//     Drive/Outputs/Out/nCtrl2 @bit 3 <-> STM Control/Control/Digital output 1
//     Drive/Outputs/Out/nDataOut2[0] <-> STM Velocity/Velocity
//   (this object) <-> Device 2 (EtherCAT)/Rack#2B-01 Coupler (EK1100)/Rack#2B-20 DR_ZF (EL7047)
//     Drive/Inputs/In/nDcOutputTime <-> InfoData/DcOutputShift
//     Drive/Inputs/In/nState1 @bit 3 <-> STM Status/Status/Error
//     Drive/Inputs/In/nState1 @bit 7 <-> STM Status/Status/Motor stall
//     Drive/Inputs/In/nState1 @bit 5 <-> STM Status/Status/Moving negative
//     Drive/Inputs/In/nState1 @bit 4 <-> STM Status/Status/Moving positive
//     Drive/Inputs/In/nState1 @bit 1 <-> STM Status/Status/Ready
//     Drive/Inputs/In/nState1 <-> STM Status/Status/Ready to enable
//     Drive/Inputs/In/nState1 @bit 6 <-> STM Status/Status/Torque reduced
//     Drive/Inputs/In/nState1 @bit 2 <-> STM Status/Status/Warning
//     Drive/Inputs/In/nState2 @bit 3 <-> STM Status/Status/Digital input 1
//     Drive/Inputs/In/nState2 @bit 4 <-> STM Status/Status/Digital input 2
//     Drive/Inputs/In/nState2 @bit 5 <-> STM Status/Status/Sync error
//     Drive/Inputs/In/nState2 @bit 7 <-> STM Status/Status/TxPDO Toggle
//     Drive/Inputs/In/nState4 @bit 1 <-> WcState/InputToggle
//     Drive/Inputs/In/nState4 <-> WcState/WcState
//     Drive/Outputs/Out/nCtrl1 <-> STM Control/Control/Enable
//     Drive/Outputs/Out/nCtrl1 @bit 2 <-> STM Control/Control/Reduce torque
//     Drive/Outputs/Out/nCtrl1 @bit 1 <-> STM Control/Control/Reset
//     Drive/Outputs/Out/nCtrl2 @bit 3 <-> STM Control/Control/Digital output 1
//     Drive/Outputs/Out/nDataOut2[0] <-> STM Velocity/Velocity
//   (this object) <-> Device 2 (EtherCAT)/B950-233-WALL-S-R01-DRL-02/EL5042_03_02-Diff-X-Y
//     Enc/Inputs/In/nComState @bit 1 <-> WcState/InputToggle
//     Enc/Inputs/In/nComState <-> WcState/WcState
//     Enc/Inputs/In/nDataIn1 <-> FB Inputs Channel 2/Position
//     Enc/Inputs/In/nDataIn1 <-> FB Inputs Channel 1/Position
//     Enc/Inputs/In/nState1 @bit 12 <-> FB Inputs Channel 2/Status/Diag
//     Enc/Inputs/In/nState1 @bit 12 <-> FB Inputs Channel 1/Status/Diag
//     Enc/Inputs/In/nState1 @bit 1 <-> FB Inputs Channel 2/Status/Error
//     Enc/Inputs/In/nState1 @bit 1 <-> FB Inputs Channel 1/Status/Error
//     Enc/Inputs/In/nState1 @bit 14 <-> FB Inputs Channel 2/Status/Input cycle counter
//     Enc/Inputs/In/nState1 @bit 14 <-> FB Inputs Channel 1/Status/Input cycle counter
//     Enc/Inputs/In/nState1 @bit 2 <-> FB Inputs Channel 2/Status/Ready
//     Enc/Inputs/In/nState1 @bit 2 <-> FB Inputs Channel 1/Status/Ready
//     Enc/Inputs/In/nState1 @bit 13 <-> FB Inputs Channel 2/Status/TxPDO State
//     Enc/Inputs/In/nState1 @bit 13 <-> FB Inputs Channel 1/Status/TxPDO State
//     Enc/Inputs/In/nState1 <-> FB Inputs Channel 2/Status/Warning
//     Enc/Inputs/In/nState1 <-> FB Inputs Channel 1/Status/Warning
//   (this object) <-> Device 2 (EtherCAT)/B950-233-WALL-S-R01-DRL-02/EL7047_03_03-Diff-Y
//     Drive/Inputs/In/nState1 @bit 3 <-> STM Status/Status/Error
//     Drive/Inputs/In/nState1 @bit 7 <-> STM Status/Status/Motor stall
//     Drive/Inputs/In/nState1 @bit 5 <-> STM Status/Status/Moving negative
//     Drive/Inputs/In/nState1 @bit 4 <-> STM Status/Status/Moving positive
//     Drive/Inputs/In/nState1 @bit 1 <-> STM Status/Status/Ready
//     Drive/Inputs/In/nState1 <-> STM Status/Status/Ready to enable
//     Drive/Inputs/In/nState1 @bit 6 <-> STM Status/Status/Torque reduced
//     Drive/Inputs/In/nState1 @bit 2 <-> STM Status/Status/Warning
//     Drive/Inputs/In/nState2 @bit 3 <-> STM Status/Status/Digital input 1
//     Drive/Inputs/In/nState2 @bit 4 <-> STM Status/Status/Digital input 2
//     Drive/Inputs/In/nState2 @bit 5 <-> STM Status/Status/Sync error
//     Drive/Inputs/In/nState2 @bit 7 <-> STM Status/Status/TxPDO Toggle
//     Drive/Inputs/In/nState4 @bit 1 <-> WcState/InputToggle
//     Drive/Inputs/In/nState4 <-> WcState/WcState
//     Drive/Outputs/Out/nCtrl1 <-> STM Control/Control/Enable
//     Drive/Outputs/Out/nCtrl1 @bit 2 <-> STM Control/Control/Reduce torque
//     Drive/Outputs/Out/nCtrl1 @bit 1 <-> STM Control/Control/Reset
//     Drive/Outputs/Out/nCtrl2 @bit 3 <-> STM Control/Control/Digital output 1
//     Drive/Outputs/Out/nDataOut2[0] <-> STM Velocity/Velocity
//   (this object) <-> Device 2 (EtherCAT)/B950-233-WALL-S-R01-DRL-02/EL5042_03_06-DIff-Z-2ThetaY
//     Enc/Inputs/In/nComState @bit 1 <-> WcState/InputToggle
//     Enc/Inputs/In/nComState <-> WcState/WcState
//     Enc/Inputs/In/nDataIn1 <-> FB Inputs Channel 1/Position
//     Enc/Inputs/In/nDataIn1 <-> FB Inputs Channel 2/Position
//     Enc/Inputs/In/nState1 @bit 12 <-> FB Inputs Channel 1/Status/Diag
//     Enc/Inputs/In/nState1 @bit 12 <-> FB Inputs Channel 2/Status/Diag
//     Enc/Inputs/In/nState1 @bit 1 <-> FB Inputs Channel 1/Status/Error
//     Enc/Inputs/In/nState1 @bit 1 <-> FB Inputs Channel 2/Status/Error
//     Enc/Inputs/In/nState1 @bit 14 <-> FB Inputs Channel 1/Status/Input cycle counter
//     Enc/Inputs/In/nState1 @bit 14 <-> FB Inputs Channel 2/Status/Input cycle counter
//     Enc/Inputs/In/nState1 @bit 2 <-> FB Inputs Channel 1/Status/Ready
//     Enc/Inputs/In/nState1 @bit 2 <-> FB Inputs Channel 2/Status/Ready
//     Enc/Inputs/In/nState1 @bit 13 <-> FB Inputs Channel 1/Status/TxPDO State
//     Enc/Inputs/In/nState1 @bit 13 <-> FB Inputs Channel 2/Status/TxPDO State
//     Enc/Inputs/In/nState1 <-> FB Inputs Channel 1/Status/Warning
//     Enc/Inputs/In/nState1 <-> FB Inputs Channel 2/Status/Warning
//   (this object) <-> Device 2 (EtherCAT)/B950-233-WALL-S-R01-DRL-02/EL7047_03_05-Diff-Z
//     Drive/Inputs/In/nState1 @bit 3 <-> STM Status/Status/Error
//     Drive/Inputs/In/nState1 @bit 7 <-> STM Status/Status/Motor stall
//     Drive/Inputs/In/nState1 @bit 5 <-> STM Status/Status/Moving negative
//     Drive/Inputs/In/nState1 @bit 4 <-> STM Status/Status/Moving positive
//     Drive/Inputs/In/nState1 @bit 1 <-> STM Status/Status/Ready
//     Drive/Inputs/In/nState1 <-> STM Status/Status/Ready to enable
//     Drive/Inputs/In/nState1 @bit 6 <-> STM Status/Status/Torque reduced
//     Drive/Inputs/In/nState1 @bit 2 <-> STM Status/Status/Warning
//     Drive/Inputs/In/nState2 @bit 3 <-> STM Status/Status/Digital input 1
//     Drive/Inputs/In/nState2 @bit 4 <-> STM Status/Status/Digital input 2
//     Drive/Inputs/In/nState2 @bit 5 <-> STM Status/Status/Sync error
//     Drive/Inputs/In/nState2 @bit 7 <-> STM Status/Status/TxPDO Toggle
//     Drive/Inputs/In/nState4 @bit 1 <-> WcState/InputToggle
//     Drive/Inputs/In/nState4 <-> WcState/WcState
//     Drive/Outputs/Out/nCtrl1 <-> STM Control/Control/Enable
//     Drive/Outputs/Out/nCtrl1 @bit 2 <-> STM Control/Control/Reduce torque
//     Drive/Outputs/Out/nCtrl1 @bit 1 <-> STM Control/Control/Reset
//     Drive/Outputs/Out/nCtrl2 @bit 3 <-> STM Control/Control/Digital output 1
//     Drive/Outputs/Out/nDataOut2[0] <-> STM Velocity/Velocity
//   (this object) <-> Device 2 (EtherCAT)/B950-233-WALL-S-R01-DRL-02/EL7047_03_07-Diff 2 Theta Y
//     Drive/Inputs/In/nState1 @bit 3 <-> STM Status/Status/Error
//     Drive/Inputs/In/nState1 @bit 7 <-> STM Status/Status/Motor stall
//     Drive/Inputs/In/nState1 @bit 5 <-> STM Status/Status/Moving negative
//     Drive/Inputs/In/nState1 @bit 4 <-> STM Status/Status/Moving positive
//     Drive/Inputs/In/nState1 @bit 1 <-> STM Status/Status/Ready
//     Drive/Inputs/In/nState1 <-> STM Status/Status/Ready to enable
//     Drive/Inputs/In/nState1 @bit 6 <-> STM Status/Status/Torque reduced
//     Drive/Inputs/In/nState1 @bit 2 <-> STM Status/Status/Warning
//     Drive/Inputs/In/nState2 @bit 3 <-> STM Status/Status/Digital input 1
//     Drive/Inputs/In/nState2 @bit 4 <-> STM Status/Status/Digital input 2
//     Drive/Inputs/In/nState2 @bit 5 <-> STM Status/Status/Sync error
//     Drive/Inputs/In/nState2 @bit 7 <-> STM Status/Status/TxPDO Toggle
//     Drive/Inputs/In/nState4 @bit 1 <-> WcState/InputToggle
//     Drive/Inputs/In/nState4 <-> WcState/WcState
//     Drive/Outputs/Out/nCtrl1 <-> STM Control/Control/Enable
//     Drive/Outputs/Out/nCtrl1 @bit 2 <-> STM Control/Control/Reduce torque
//     Drive/Outputs/Out/nCtrl1 @bit 1 <-> STM Control/Control/Reset
//     Drive/Outputs/Out/nCtrl2 @bit 3 <-> STM Control/Control/Digital output 1
//     Drive/Outputs/Out/nDataOut2[0] <-> STM Velocity/Velocity
//   (this object) <-> Device 2 (EtherCAT)/B950-233-WALL-S-R01-DRL-02/EL5042_03_13 - Diff - Phi - Chi
//     Enc/Inputs/In/nComState @bit 1 <-> WcState/InputToggle
//     Enc/Inputs/In/nComState <-> WcState/WcState
//     Enc/Inputs/In/nDataIn1 <-> FB Inputs Channel 1/Position
//     Enc/Inputs/In/nDataIn1 <-> FB Inputs Channel 2/Position
//     Enc/Inputs/In/nState1 @bit 12 <-> FB Inputs Channel 1/Status/Diag
//     Enc/Inputs/In/nState1 @bit 12 <-> FB Inputs Channel 2/Status/Diag
//     Enc/Inputs/In/nState1 @bit 1 <-> FB Inputs Channel 1/Status/Error
//     Enc/Inputs/In/nState1 @bit 1 <-> FB Inputs Channel 2/Status/Error
//     Enc/Inputs/In/nState1 @bit 14 <-> FB Inputs Channel 1/Status/Input cycle counter
//     Enc/Inputs/In/nState1 @bit 14 <-> FB Inputs Channel 2/Status/Input cycle counter
//     Enc/Inputs/In/nState1 @bit 2 <-> FB Inputs Channel 1/Status/Ready
//     Enc/Inputs/In/nState1 @bit 2 <-> FB Inputs Channel 2/Status/Ready
//     Enc/Inputs/In/nState1 @bit 13 <-> FB Inputs Channel 1/Status/TxPDO State
//     Enc/Inputs/In/nState1 @bit 13 <-> FB Inputs Channel 2/Status/TxPDO State
//     Enc/Inputs/In/nState1 <-> FB Inputs Channel 1/Status/Warning
//     Enc/Inputs/In/nState1 <-> FB Inputs Channel 2/Status/Warning
//   (this object) <-> Device 2 (EtherCAT)/B950-233-WALL-S-R01-DRL-02/EL7047_03_12-Diff - Phi
//     Drive/Inputs/In/nState1 @bit 3 <-> STM Status/Status/Error
//     Drive/Inputs/In/nState1 @bit 7 <-> STM Status/Status/Motor stall
//     Drive/Inputs/In/nState1 @bit 5 <-> STM Status/Status/Moving negative
//     Drive/Inputs/In/nState1 @bit 4 <-> STM Status/Status/Moving positive
//     Drive/Inputs/In/nState1 @bit 1 <-> STM Status/Status/Ready
//     Drive/Inputs/In/nState1 <-> STM Status/Status/Ready to enable
//     Drive/Inputs/In/nState1 @bit 6 <-> STM Status/Status/Torque reduced
//     Drive/Inputs/In/nState1 @bit 2 <-> STM Status/Status/Warning
//     Drive/Inputs/In/nState2 @bit 3 <-> STM Status/Status/Digital input 1
//     Drive/Inputs/In/nState2 @bit 4 <-> STM Status/Status/Digital input 2
//     Drive/Inputs/In/nState2 @bit 5 <-> STM Status/Status/Sync error
//     Drive/Inputs/In/nState2 @bit 7 <-> STM Status/Status/TxPDO Toggle
//     Drive/Inputs/In/nState4 @bit 1 <-> WcState/InputToggle
//     Drive/Inputs/In/nState4 <-> WcState/WcState
//     Drive/Outputs/Out/nCtrl1 <-> STM Control/Control/Enable
//     Drive/Outputs/Out/nCtrl1 @bit 2 <-> STM Control/Control/Reduce torque
//     Drive/Outputs/Out/nCtrl1 @bit 1 <-> STM Control/Control/Reset
//     Drive/Outputs/Out/nCtrl2 @bit 3 <-> STM Control/Control/Digital output 1
//     Drive/Outputs/Out/nDataOut2[0] <-> STM Velocity/Velocity
//   (this object) <-> Device 2 (EtherCAT)/B950-233-WALL-S-R01-DRL-02/EL7047_03_14-Diff - Chi
//     Drive/Inputs/In/nState1 @bit 3 <-> STM Status/Status/Error
//     Drive/Inputs/In/nState1 @bit 7 <-> STM Status/Status/Motor stall
//     Drive/Inputs/In/nState1 @bit 5 <-> STM Status/Status/Moving negative
//     Drive/Inputs/In/nState1 @bit 4 <-> STM Status/Status/Moving positive
//     Drive/Inputs/In/nState1 @bit 1 <-> STM Status/Status/Ready
//     Drive/Inputs/In/nState1 <-> STM Status/Status/Ready to enable
//     Drive/Inputs/In/nState1 @bit 6 <-> STM Status/Status/Torque reduced
//     Drive/Inputs/In/nState1 @bit 2 <-> STM Status/Status/Warning
//     Drive/Inputs/In/nState2 @bit 3 <-> STM Status/Status/Digital input 1
//     Drive/Inputs/In/nState2 @bit 4 <-> STM Status/Status/Digital input 2
//     Drive/Inputs/In/nState2 @bit 5 <-> STM Status/Status/Sync error
//     Drive/Inputs/In/nState2 @bit 7 <-> STM Status/Status/TxPDO Toggle
//     Drive/Inputs/In/nState4 @bit 1 <-> WcState/InputToggle
//     Drive/Inputs/In/nState4 <-> WcState/WcState
//     Drive/Outputs/Out/nCtrl1 <-> STM Control/Control/Enable
//     Drive/Outputs/Out/nCtrl1 @bit 2 <-> STM Control/Control/Reduce torque
//     Drive/Outputs/Out/nCtrl1 @bit 1 <-> STM Control/Control/Reset
//     Drive/Outputs/Out/nCtrl2 @bit 3 <-> STM Control/Control/Digital output 1
//     Drive/Outputs/Out/nDataOut2[0] <-> STM Velocity/Velocity
//   (this object) <-> Device 2 (EtherCAT)/B950-233-WALL-S-R01-DRL-02/EL5042_03_17 - Diff - Theta - 2Theta
//     Enc/Inputs/In/nComState @bit 1 <-> WcState/InputToggle
//     Enc/Inputs/In/nComState <-> WcState/WcState
//     Enc/Inputs/In/nDataIn1 <-> FB Inputs Channel 2/Position
//     Enc/Inputs/In/nState1 @bit 12 <-> FB Inputs Channel 2/Status/Diag
//     Enc/Inputs/In/nState1 @bit 12 <-> FB Inputs Channel 1/Status/Diag
//     Enc/Inputs/In/nState1 @bit 1 <-> FB Inputs Channel 2/Status/Error
//     Enc/Inputs/In/nState1 @bit 1 <-> FB Inputs Channel 1/Status/Error
//     Enc/Inputs/In/nState1 @bit 14 <-> FB Inputs Channel 2/Status/Input cycle counter
//     Enc/Inputs/In/nState1 @bit 14 <-> FB Inputs Channel 1/Status/Input cycle counter
//     Enc/Inputs/In/nState1 @bit 2 <-> FB Inputs Channel 2/Status/Ready
//     Enc/Inputs/In/nState1 @bit 2 <-> FB Inputs Channel 1/Status/Ready
//     Enc/Inputs/In/nState1 @bit 13 <-> FB Inputs Channel 2/Status/TxPDO State
//     Enc/Inputs/In/nState1 @bit 13 <-> FB Inputs Channel 1/Status/TxPDO State
//     Enc/Inputs/In/nState1 <-> FB Inputs Channel 2/Status/Warning
//     Enc/Inputs/In/nState1 <-> FB Inputs Channel 1/Status/Warning
//   (this object) <-> Device 2 (EtherCAT)/B950-233-WALL-S-R01-DRL-02/EL7047_03_18 - Diff - 2Theta
//     Drive/Inputs/In/nState1 @bit 3 <-> STM Status/Status/Error
//     Drive/Inputs/In/nState1 @bit 7 <-> STM Status/Status/Motor stall
//     Drive/Inputs/In/nState1 @bit 5 <-> STM Status/Status/Moving negative
//     Drive/Inputs/In/nState1 @bit 4 <-> STM Status/Status/Moving positive
//     Drive/Inputs/In/nState1 @bit 1 <-> STM Status/Status/Ready
//     Drive/Inputs/In/nState1 <-> STM Status/Status/Ready to enable
//     Drive/Inputs/In/nState1 @bit 6 <-> STM Status/Status/Torque reduced
//     Drive/Inputs/In/nState1 @bit 2 <-> STM Status/Status/Warning
//     Drive/Inputs/In/nState2 @bit 3 <-> STM Status/Status/Digital input 1
//     Drive/Inputs/In/nState2 @bit 4 <-> STM Status/Status/Digital input 2
//     Drive/Inputs/In/nState2 @bit 5 <-> STM Status/Status/Sync error
//     Drive/Inputs/In/nState2 @bit 7 <-> STM Status/Status/TxPDO Toggle
//     Drive/Inputs/In/nState4 @bit 1 <-> WcState/InputToggle
//     Drive/Inputs/In/nState4 <-> WcState/WcState
//     Drive/Outputs/Out/nCtrl1 <-> STM Control/Control/Enable
//     Drive/Outputs/Out/nCtrl1 @bit 2 <-> STM Control/Control/Reduce torque
//     Drive/Outputs/Out/nCtrl1 @bit 1 <-> STM Control/Control/Reset
//     Drive/Outputs/Out/nCtrl2 @bit 3 <-> STM Control/Control/Digital output 1
//     Drive/Outputs/Out/nDataOut2[0] <-> STM Velocity/Velocity
//   (this object) <-> Device 2 (EtherCAT)/B950-233-WALL-S-R01-DRL-02/EL7047_03_16 - Diff - Theta
//     Drive/Inputs/In/nState1 @bit 3 <-> STM Status/Status/Error
//     Drive/Inputs/In/nState1 @bit 7 <-> STM Status/Status/Motor stall
//     Drive/Inputs/In/nState1 @bit 5 <-> STM Status/Status/Moving negative
//     Drive/Inputs/In/nState1 @bit 4 <-> STM Status/Status/Moving positive
//     Drive/Inputs/In/nState1 @bit 1 <-> STM Status/Status/Ready
//     Drive/Inputs/In/nState1 <-> STM Status/Status/Ready to enable
//     Drive/Inputs/In/nState1 @bit 6 <-> STM Status/Status/Torque reduced
//     Drive/Inputs/In/nState1 @bit 2 <-> STM Status/Status/Warning
//     Drive/Inputs/In/nState2 @bit 3 <-> STM Status/Status/Digital input 1
//     Drive/Inputs/In/nState2 @bit 4 <-> STM Status/Status/Digital input 2
//     Drive/Inputs/In/nState2 @bit 5 <-> STM Status/Status/Sync error
//     Drive/Inputs/In/nState2 @bit 7 <-> STM Status/Status/TxPDO Toggle
//     Drive/Inputs/In/nState4 @bit 1 <-> WcState/InputToggle
//     Drive/Inputs/In/nState4 <-> WcState/WcState
//     Drive/Outputs/Out/nCtrl1 <-> STM Control/Control/Enable
//     Drive/Outputs/Out/nCtrl1 @bit 2 <-> STM Control/Control/Reduce torque
//     Drive/Outputs/Out/nCtrl1 @bit 1 <-> STM Control/Control/Reset
//     Drive/Outputs/Out/nCtrl2 @bit 3 <-> STM Control/Control/Digital output 1
//     Drive/Outputs/Out/nDataOut2[0] <-> STM Velocity/Velocity
//   (this object) <-> Device 2 (EtherCAT)/B950-233-WALL-S-R01-DRL-02/EL7047_03_01-Diff-X
//     Drive/Inputs/In/nState1 @bit 3 <-> STM Status/Status/Error
//     Drive/Inputs/In/nState1 @bit 7 <-> STM Status/Status/Motor stall
//     Drive/Inputs/In/nState1 @bit 5 <-> STM Status/Status/Moving negative
//     Drive/Inputs/In/nState1 @bit 4 <-> STM Status/Status/Moving positive
//     Drive/Inputs/In/nState1 @bit 1 <-> STM Status/Status/Ready
//     Drive/Inputs/In/nState1 <-> STM Status/Status/Ready to enable
//     Drive/Inputs/In/nState1 @bit 6 <-> STM Status/Status/Torque reduced
//     Drive/Inputs/In/nState1 @bit 2 <-> STM Status/Status/Warning
//     Drive/Inputs/In/nState2 @bit 3 <-> STM Status/Status/Digital input 1
//     Drive/Inputs/In/nState2 @bit 4 <-> STM Status/Status/Digital input 2
//     Drive/Inputs/In/nState2 @bit 5 <-> STM Status/Status/Sync error
//     Drive/Inputs/In/nState2 @bit 7 <-> STM Status/Status/TxPDO Toggle
//     Drive/Inputs/In/nState4 @bit 1 <-> WcState/InputToggle
//     Drive/Inputs/In/nState4 <-> WcState/WcState
//     Drive/Outputs/Out/nCtrl1 <-> STM Control/Control/Enable
//     Drive/Outputs/Out/nCtrl1 @bit 2 <-> STM Control/Control/Reduce torque
//     Drive/Outputs/Out/nCtrl1 @bit 1 <-> STM Control/Control/Reset
//     Drive/Outputs/Out/nCtrl2 @bit 3 <-> STM Control/Control/Digital output 1
//     Drive/Outputs/Out/nDataOut2[0] <-> STM Velocity/Velocity
//   (this object) <-> Device 2 (EtherCAT)/B950-233-WALL-S-R01-DRL-01/EL5042_02_05 - LAS_VIS
//     Enc/Inputs/In/nComState @bit 1 <-> WcState/InputToggle
//     Enc/Inputs/In/nComState <-> WcState/WcState
//     Enc/Inputs/In/nDataIn1 <-> FB Inputs Channel 1/Position
//     Enc/Inputs/In/nState1 @bit 12 <-> FB Inputs Channel 1/Status/Diag
//     Enc/Inputs/In/nState1 @bit 1 <-> FB Inputs Channel 1/Status/Error
//     Enc/Inputs/In/nState1 @bit 14 <-> FB Inputs Channel 1/Status/Input cycle counter
//     Enc/Inputs/In/nState1 @bit 2 <-> FB Inputs Channel 1/Status/Ready
//     Enc/Inputs/In/nState1 @bit 13 <-> FB Inputs Channel 1/Status/TxPDO State
//     Enc/Inputs/In/nState1 <-> FB Inputs Channel 1/Status/Warning
//   (this object) <-> Device 2 (EtherCAT)/B950-233-WALL-S-R01-DRL-01/EL7031_02_04 - LAS_VIS
//     Drive/Inputs/In/nState1 @bit 3 <-> STM Status/Status/Error
//     Drive/Inputs/In/nState1 @bit 5 <-> STM Status/Status/Moving negative
//     Drive/Inputs/In/nState1 @bit 4 <-> STM Status/Status/Moving positive
//     Drive/Inputs/In/nState1 @bit 1 <-> STM Status/Status/Ready
//     Drive/Inputs/In/nState1 <-> STM Status/Status/Ready to enable
//     Drive/Inputs/In/nState1 @bit 6 <-> STM Status/Status/Torque reduced
//     Drive/Inputs/In/nState1 @bit 2 <-> STM Status/Status/Warning
//     Drive/Inputs/In/nState2 @bit 3 <-> STM Status/Status/Digital input 1
//     Drive/Inputs/In/nState2 @bit 4 <-> STM Status/Status/Digital input 2
//     Drive/Inputs/In/nState2 @bit 5 <-> STM Status/Status/Sync error
//     Drive/Inputs/In/nState2 @bit 7 <-> STM Status/Status/TxPDO Toggle
//     Drive/Inputs/In/nState4 @bit 1 <-> WcState/InputToggle
//     Drive/Inputs/In/nState4 <-> WcState/WcState
//     Drive/Outputs/Out/nCtrl1 <-> STM Control/Control/Enable
//     Drive/Outputs/Out/nCtrl1 @bit 2 <-> STM Control/Control/Reduce torque
//     Drive/Outputs/Out/nCtrl1 @bit 1 <-> STM Control/Control/Reset
//     Drive/Outputs/Out/nDataOut2[0] <-> STM Velocity/Velocity
//   (this object) <-> Device 2 (EtherCAT)/B950-233-WALL-S-R01-DRL-01/EL5042_02_08 - LAS_D_V-H
//     Enc/Inputs/In/nComState @bit 1 <-> WcState/InputToggle
//     Enc/Inputs/In/nComState <-> WcState/WcState
//     Enc/Inputs/In/nDataIn1 <-> FB Inputs Channel 2/Position
//     Enc/Inputs/In/nDataIn1 <-> FB Inputs Channel 1/Position
//     Enc/Inputs/In/nState1 @bit 12 <-> FB Inputs Channel 2/Status/Diag
//     Enc/Inputs/In/nState1 @bit 12 <-> FB Inputs Channel 1/Status/Diag
//     Enc/Inputs/In/nState1 @bit 1 <-> FB Inputs Channel 2/Status/Error
//     Enc/Inputs/In/nState1 @bit 1 <-> FB Inputs Channel 1/Status/Error
//     Enc/Inputs/In/nState1 @bit 14 <-> FB Inputs Channel 2/Status/Input cycle counter
//     Enc/Inputs/In/nState1 @bit 14 <-> FB Inputs Channel 1/Status/Input cycle counter
//     Enc/Inputs/In/nState1 @bit 2 <-> FB Inputs Channel 2/Status/Ready
//     Enc/Inputs/In/nState1 @bit 2 <-> FB Inputs Channel 1/Status/Ready
//     Enc/Inputs/In/nState1 @bit 13 <-> FB Inputs Channel 2/Status/TxPDO State
//     Enc/Inputs/In/nState1 @bit 13 <-> FB Inputs Channel 1/Status/TxPDO State
//     Enc/Inputs/In/nState1 <-> FB Inputs Channel 2/Status/Warning
//     Enc/Inputs/In/nState1 <-> FB Inputs Channel 1/Status/Warning
//   (this object) <-> Device 2 (EtherCAT)/B950-233-WALL-S-R01-DRL-01/EL7031_02_07 - LAS_D_H
//     Drive/Inputs/In/nState1 @bit 3 <-> STM Status/Status/Error
//     Drive/Inputs/In/nState1 @bit 5 <-> STM Status/Status/Moving negative
//     Drive/Inputs/In/nState1 @bit 4 <-> STM Status/Status/Moving positive
//     Drive/Inputs/In/nState1 @bit 1 <-> STM Status/Status/Ready
//     Drive/Inputs/In/nState1 <-> STM Status/Status/Ready to enable
//     Drive/Inputs/In/nState1 @bit 6 <-> STM Status/Status/Torque reduced
//     Drive/Inputs/In/nState1 @bit 2 <-> STM Status/Status/Warning
//     Drive/Inputs/In/nState2 @bit 3 <-> STM Status/Status/Digital input 1
//     Drive/Inputs/In/nState2 @bit 4 <-> STM Status/Status/Digital input 2
//     Drive/Inputs/In/nState2 @bit 5 <-> STM Status/Status/Sync error
//     Drive/Inputs/In/nState2 @bit 7 <-> STM Status/Status/TxPDO Toggle
//     Drive/Inputs/In/nState4 @bit 1 <-> WcState/InputToggle
//     Drive/Inputs/In/nState4 <-> WcState/WcState
//     Drive/Outputs/Out/nCtrl1 <-> STM Control/Control/Enable
//     Drive/Outputs/Out/nCtrl1 @bit 2 <-> STM Control/Control/Reduce torque
//     Drive/Outputs/Out/nCtrl1 @bit 1 <-> STM Control/Control/Reset
//     Drive/Outputs/Out/nDataOut2[0] <-> STM Velocity/Velocity
//   (this object) <-> Device 2 (EtherCAT)/B950-233-WALL-S-R01-DRL-01/EL7031_02_09 - LAS_D_V
//     Drive/Inputs/In/nState1 @bit 3 <-> STM Status/Status/Error
//     Drive/Inputs/In/nState1 @bit 5 <-> STM Status/Status/Moving negative
//     Drive/Inputs/In/nState1 @bit 4 <-> STM Status/Status/Moving positive
//     Drive/Inputs/In/nState1 @bit 1 <-> STM Status/Status/Ready
//     Drive/Inputs/In/nState1 <-> STM Status/Status/Ready to enable
//     Drive/Inputs/In/nState1 @bit 6 <-> STM Status/Status/Torque reduced
//     Drive/Inputs/In/nState1 @bit 2 <-> STM Status/Status/Warning
//     Drive/Inputs/In/nState2 @bit 3 <-> STM Status/Status/Digital input 1
//     Drive/Inputs/In/nState2 @bit 4 <-> STM Status/Status/Digital input 2
//     Drive/Inputs/In/nState2 @bit 5 <-> STM Status/Status/Sync error
//     Drive/Inputs/In/nState2 @bit 7 <-> STM Status/Status/TxPDO Toggle
//     Drive/Inputs/In/nState4 @bit 1 <-> WcState/InputToggle
//     Drive/Inputs/In/nState4 <-> WcState/WcState
//     Drive/Outputs/Out/nCtrl1 <-> STM Control/Control/Enable
//     Drive/Outputs/Out/nCtrl1 @bit 2 <-> STM Control/Control/Reduce torque
//     Drive/Outputs/Out/nCtrl1 @bit 1 <-> STM Control/Control/Reset
//     Drive/Outputs/Out/nDataOut2[0] <-> STM Velocity/Velocity
//   (this object) <-> Device 2 (EtherCAT)/B950-233-WALL-S-R01-DRL-03_SDS/EL5042_04_02
//     Enc/Inputs/In/nComState @bit 1 <-> WcState/InputToggle
//     Enc/Inputs/In/nComState <-> WcState/WcState
//     Enc/Inputs/In/nDataIn1 <-> FB Inputs Channel 1/Position
//     Enc/Inputs/In/nDataIn1 <-> FB Inputs Channel 2/Position
//     Enc/Inputs/In/nState1 @bit 12 <-> FB Inputs Channel 1/Status/Diag
//     Enc/Inputs/In/nState1 @bit 12 <-> FB Inputs Channel 2/Status/Diag
//     Enc/Inputs/In/nState1 @bit 1 <-> FB Inputs Channel 1/Status/Error
//     Enc/Inputs/In/nState1 @bit 1 <-> FB Inputs Channel 2/Status/Error
//     Enc/Inputs/In/nState1 @bit 14 <-> FB Inputs Channel 1/Status/Input cycle counter
//     Enc/Inputs/In/nState1 @bit 14 <-> FB Inputs Channel 2/Status/Input cycle counter
//     Enc/Inputs/In/nState1 @bit 2 <-> FB Inputs Channel 1/Status/Ready
//     Enc/Inputs/In/nState1 @bit 2 <-> FB Inputs Channel 2/Status/Ready
//     Enc/Inputs/In/nState1 @bit 13 <-> FB Inputs Channel 1/Status/TxPDO State
//     Enc/Inputs/In/nState1 @bit 13 <-> FB Inputs Channel 2/Status/TxPDO State
//     Enc/Inputs/In/nState1 <-> FB Inputs Channel 1/Status/Warning
//     Enc/Inputs/In/nState1 <-> FB Inputs Channel 2/Status/Warning
//   (this object) <-> Device 2 (EtherCAT)/B950-233-WALL-S-R01-DRL-03_SDS/EL7047_04_01
//     Drive/Inputs/In/nState1 @bit 3 <-> STM Status/Status/Error
//     Drive/Inputs/In/nState1 @bit 7 <-> STM Status/Status/Motor stall
//     Drive/Inputs/In/nState1 @bit 5 <-> STM Status/Status/Moving negative
//     Drive/Inputs/In/nState1 @bit 4 <-> STM Status/Status/Moving positive
//     Drive/Inputs/In/nState1 @bit 1 <-> STM Status/Status/Ready
//     Drive/Inputs/In/nState1 <-> STM Status/Status/Ready to enable
//     Drive/Inputs/In/nState1 @bit 6 <-> STM Status/Status/Torque reduced
//     Drive/Inputs/In/nState1 @bit 2 <-> STM Status/Status/Warning
//     Drive/Inputs/In/nState2 @bit 3 <-> STM Status/Status/Digital input 1
//     Drive/Inputs/In/nState2 @bit 4 <-> STM Status/Status/Digital input 2
//     Drive/Inputs/In/nState2 @bit 5 <-> STM Status/Status/Sync error
//     Drive/Inputs/In/nState2 @bit 7 <-> STM Status/Status/TxPDO Toggle
//     Drive/Inputs/In/nState4 @bit 1 <-> WcState/InputToggle
//     Drive/Inputs/In/nState4 <-> WcState/WcState
//     Drive/Outputs/Out/nCtrl1 <-> STM Control/Control/Enable
//     Drive/Outputs/Out/nCtrl1 @bit 2 <-> STM Control/Control/Reduce torque
//     Drive/Outputs/Out/nCtrl1 @bit 1 <-> STM Control/Control/Reset
//     Drive/Outputs/Out/nCtrl2 @bit 3 <-> STM Control/Control/Digital output 1
//     Drive/Outputs/Out/nDataOut2[0] <-> STM Velocity/Velocity
//   (this object) <-> Device 2 (EtherCAT)/B950-233-WALL-S-R01-DRL-03_SDS/EL7047_04_03
//     Drive/Inputs/In/nState1 @bit 3 <-> STM Status/Status/Error
//     Drive/Inputs/In/nState1 @bit 7 <-> STM Status/Status/Motor stall
//     Drive/Inputs/In/nState1 @bit 5 <-> STM Status/Status/Moving negative
//     Drive/Inputs/In/nState1 @bit 4 <-> STM Status/Status/Moving positive
//     Drive/Inputs/In/nState1 @bit 1 <-> STM Status/Status/Ready
//     Drive/Inputs/In/nState1 <-> STM Status/Status/Ready to enable
//     Drive/Inputs/In/nState1 @bit 6 <-> STM Status/Status/Torque reduced
//     Drive/Inputs/In/nState1 @bit 2 <-> STM Status/Status/Warning
//     Drive/Inputs/In/nState2 @bit 3 <-> STM Status/Status/Digital input 1
//     Drive/Inputs/In/nState2 @bit 4 <-> STM Status/Status/Digital input 2
//     Drive/Inputs/In/nState2 @bit 5 <-> STM Status/Status/Sync error
//     Drive/Inputs/In/nState2 @bit 7 <-> STM Status/Status/TxPDO Toggle
//     Drive/Inputs/In/nState4 @bit 1 <-> WcState/InputToggle
//     Drive/Inputs/In/nState4 <-> WcState/WcState
//     Drive/Outputs/Out/nCtrl1 <-> STM Control/Control/Enable
//     Drive/Outputs/Out/nCtrl1 @bit 2 <-> STM Control/Control/Reduce torque
//     Drive/Outputs/Out/nCtrl1 @bit 1 <-> STM Control/Control/Reset
//     Drive/Outputs/Out/nCtrl2 @bit 3 <-> STM Control/Control/Digital output 1
//     Drive/Outputs/Out/nDataOut2[0] <-> STM Velocity/Velocity
//   (this object) <-> Device 2 (EtherCAT)/B950-233-WALL-S-R01-DRL-03_SDS/EL5042_04_06
//     Enc/Inputs/In/nComState @bit 1 <-> WcState/InputToggle
//     Enc/Inputs/In/nComState <-> WcState/WcState
//     Enc/Inputs/In/nDataIn1 <-> FB Inputs Channel 1/Position
//     Enc/Inputs/In/nState1 @bit 12 <-> FB Inputs Channel 1/Status/Diag
//     Enc/Inputs/In/nState1 @bit 1 <-> FB Inputs Channel 1/Status/Error
//     Enc/Inputs/In/nState1 @bit 14 <-> FB Inputs Channel 1/Status/Input cycle counter
//     Enc/Inputs/In/nState1 @bit 2 <-> FB Inputs Channel 1/Status/Ready
//     Enc/Inputs/In/nState1 @bit 13 <-> FB Inputs Channel 1/Status/TxPDO State
//     Enc/Inputs/In/nState1 <-> FB Inputs Channel 1/Status/Warning
//   (this object) <-> Device 2 (EtherCAT)/B950-233-WALL-S-R01-DRL-03_SDS/EL7047_04_05
//     Drive/Inputs/In/nState1 @bit 3 <-> STM Status/Status/Error
//     Drive/Inputs/In/nState1 @bit 7 <-> STM Status/Status/Motor stall
//     Drive/Inputs/In/nState1 @bit 5 <-> STM Status/Status/Moving negative
//     Drive/Inputs/In/nState1 @bit 4 <-> STM Status/Status/Moving positive
//     Drive/Inputs/In/nState1 @bit 1 <-> STM Status/Status/Ready
//     Drive/Inputs/In/nState1 <-> STM Status/Status/Ready to enable
//     Drive/Inputs/In/nState1 @bit 6 <-> STM Status/Status/Torque reduced
//     Drive/Inputs/In/nState1 @bit 2 <-> STM Status/Status/Warning
//     Drive/Inputs/In/nState2 @bit 3 <-> STM Status/Status/Digital input 1
//     Drive/Inputs/In/nState2 @bit 4 <-> STM Status/Status/Digital input 2
//     Drive/Inputs/In/nState2 @bit 5 <-> STM Status/Status/Sync error
//     Drive/Inputs/In/nState2 @bit 7 <-> STM Status/Status/TxPDO Toggle
//     Drive/Inputs/In/nState4 @bit 1 <-> WcState/InputToggle
//     Drive/Inputs/In/nState4 <-> WcState/WcState
//     Drive/Outputs/Out/nCtrl1 <-> STM Control/Control/Enable
//     Drive/Outputs/Out/nCtrl1 @bit 2 <-> STM Control/Control/Reduce torque
//     Drive/Outputs/Out/nCtrl1 @bit 1 <-> STM Control/Control/Reset
//     Drive/Outputs/Out/nCtrl2 @bit 3 <-> STM Control/Control/Digital output 1
//     Drive/Outputs/Out/nDataOut2[0] <-> STM Velocity/Velocity
//   (this object) <-> Device 2 (EtherCAT)/B950-233-WALL-S-R01-DRL-03_SDS/EK1122_04_17/B950-233-K2S13-DRL-01/EL5101_05_01
//     Enc/Inputs/In/nDataIn1[0] <-> ENC Status compact/Counter value
//     Enc/Inputs/In/nDataIn2[0] <-> ENC Status compact/Latch value
//     Enc/Inputs/In/nState1 @bit 4 <-> ENC Status compact/Status/Counter overflow
//     Enc/Inputs/In/nState1 @bit 3 <-> ENC Status compact/Status/Counter underflow
//     Enc/Inputs/In/nState1 @bit 7 <-> ENC Status compact/Status/Extrapolation stall
//     Enc/Inputs/In/nState1 <-> ENC Status compact/Status/Latch C valid
//     Enc/Inputs/In/nState1 @bit 1 <-> ENC Status compact/Status/Latch extern valid
//     Enc/Inputs/In/nState1 @bit 6 <-> ENC Status compact/Status/Open circuit
//     Enc/Inputs/In/nState1 @bit 2 <-> ENC Status compact/Status/Set counter done
//     Enc/Inputs/In/nState1 @bit 5 <-> ENC Status compact/Status/Status of input status
//     Enc/Inputs/In/nState2 @bit 4 <-> ENC Status compact/Status/Status of extern latch
//     Enc/Inputs/In/nState2 <-> ENC Status compact/Status/Status of input A
//     Enc/Inputs/In/nState2 @bit 1 <-> ENC Status compact/Status/Status of input B
//     Enc/Inputs/In/nState2 @bit 2 <-> ENC Status compact/Status/Status of input C
//     Enc/Inputs/In/nState2 @bit 3 <-> ENC Status compact/Status/Status of input gate
//     Enc/Inputs/In/nState2 @bit 5 <-> ENC Status compact/Status/Sync error
//     Enc/Inputs/In/nState2 @bit 6 <-> ENC Status compact/Status/TxPDO State
//     Enc/Inputs/In/nState2 @bit 7 <-> ENC Status compact/Status/TxPDO Toggle
//     Enc/Inputs/In/nState4 @bit 1 <-> WcState/InputToggle
//     Enc/Inputs/In/nState4 <-> WcState/WcState
//     Enc/Outputs/Out/nCtrl1 <-> ENC Control compact/Control/Enable latch C
//     Enc/Outputs/Out/nCtrl1 @bit 3 <-> ENC Control compact/Control/Enable latch extern on negative edge
//     Enc/Outputs/Out/nCtrl1 @bit 1 <-> ENC Control compact/Control/Enable latch extern on positive edge
//     Enc/Outputs/Out/nCtrl1 @bit 2 <-> ENC Control compact/Control/Set counter
//     Enc/Outputs/Out/nDataOut1[0] <-> ENC Control compact/Set counter value
//   (this object) <-> Device 2 (EtherCAT)/B950-233-WALL-S-R01-DRL-03_SDS/EL7047_04_07
//     Drive/Inputs/In/nState1 @bit 3 <-> STM Status/Status/Error
//     Drive/Inputs/In/nState1 @bit 7 <-> STM Status/Status/Motor stall
//     Drive/Inputs/In/nState1 @bit 5 <-> STM Status/Status/Moving negative
//     Drive/Inputs/In/nState1 @bit 4 <-> STM Status/Status/Moving positive
//     Drive/Inputs/In/nState1 @bit 1 <-> STM Status/Status/Ready
//     Drive/Inputs/In/nState1 <-> STM Status/Status/Ready to enable
//     Drive/Inputs/In/nState1 @bit 6 <-> STM Status/Status/Torque reduced
//     Drive/Inputs/In/nState1 @bit 2 <-> STM Status/Status/Warning
//     Drive/Inputs/In/nState2 @bit 3 <-> STM Status/Status/Digital input 1
//     Drive/Inputs/In/nState2 @bit 4 <-> STM Status/Status/Digital input 2
//     Drive/Inputs/In/nState2 @bit 5 <-> STM Status/Status/Sync error
//     Drive/Inputs/In/nState2 @bit 7 <-> STM Status/Status/TxPDO Toggle
//     Drive/Inputs/In/nState4 @bit 1 <-> WcState/InputToggle
//     Drive/Inputs/In/nState4 <-> WcState/WcState
//     Drive/Outputs/Out/nCtrl1 <-> STM Control/Control/Enable
//     Drive/Outputs/Out/nCtrl1 @bit 2 <-> STM Control/Control/Reduce torque
//     Drive/Outputs/Out/nCtrl1 @bit 1 <-> STM Control/Control/Reset
//     Drive/Outputs/Out/nCtrl2 @bit 3 <-> STM Control/Control/Digital output 1
//     Drive/Outputs/Out/nDataOut2[0] <-> STM Velocity/Velocity
//   (this object) <-> Device 2 (EtherCAT)/B950-233-WALL-S-R01-DRL-03_SDS/EK1122_04_17/B950-233-K2S13-DRL-01/EL5101_05_02
//     Enc/Inputs/In/nDataIn1[0] <-> ENC Status compact/Counter value
//     Enc/Inputs/In/nDataIn2[0] <-> ENC Status compact/Latch value
//     Enc/Inputs/In/nState1 @bit 4 <-> ENC Status compact/Status/Counter overflow
//     Enc/Inputs/In/nState1 @bit 3 <-> ENC Status compact/Status/Counter underflow
//     Enc/Inputs/In/nState1 @bit 7 <-> ENC Status compact/Status/Extrapolation stall
//     Enc/Inputs/In/nState1 <-> ENC Status compact/Status/Latch C valid
//     Enc/Inputs/In/nState1 @bit 1 <-> ENC Status compact/Status/Latch extern valid
//     Enc/Inputs/In/nState1 @bit 6 <-> ENC Status compact/Status/Open circuit
//     Enc/Inputs/In/nState1 @bit 2 <-> ENC Status compact/Status/Set counter done
//     Enc/Inputs/In/nState1 @bit 5 <-> ENC Status compact/Status/Status of input status
//     Enc/Inputs/In/nState2 @bit 4 <-> ENC Status compact/Status/Status of extern latch
//     Enc/Inputs/In/nState2 <-> ENC Status compact/Status/Status of input A
//     Enc/Inputs/In/nState2 @bit 1 <-> ENC Status compact/Status/Status of input B
//     Enc/Inputs/In/nState2 @bit 2 <-> ENC Status compact/Status/Status of input C
//     Enc/Inputs/In/nState2 @bit 3 <-> ENC Status compact/Status/Status of input gate
//     Enc/Inputs/In/nState2 @bit 5 <-> ENC Status compact/Status/Sync error
//     Enc/Inputs/In/nState2 @bit 6 <-> ENC Status compact/Status/TxPDO State
//     Enc/Inputs/In/nState2 @bit 7 <-> ENC Status compact/Status/TxPDO Toggle
//     Enc/Inputs/In/nState4 @bit 1 <-> WcState/InputToggle
//     Enc/Inputs/In/nState4 <-> WcState/WcState
//     Enc/Outputs/Out/nCtrl1 <-> ENC Control compact/Control/Enable latch C
//     Enc/Outputs/Out/nCtrl1 @bit 3 <-> ENC Control compact/Control/Enable latch extern on negative edge
//     Enc/Outputs/Out/nCtrl1 @bit 1 <-> ENC Control compact/Control/Enable latch extern on positive edge
//     Enc/Outputs/Out/nCtrl1 @bit 2 <-> ENC Control compact/Control/Set counter
//     Enc/Outputs/Out/nDataOut1[0] <-> ENC Control compact/Set counter value
//   (this object) <-> Device 2 (EtherCAT)/B950-233-WALL-S-R01-DRL-03_SDS/EL7047_04_10
//     Drive/Inputs/In/nState1 @bit 3 <-> STM Status/Status/Error
//     Drive/Inputs/In/nState1 @bit 7 <-> STM Status/Status/Motor stall
//     Drive/Inputs/In/nState1 @bit 5 <-> STM Status/Status/Moving negative
//     Drive/Inputs/In/nState1 @bit 4 <-> STM Status/Status/Moving positive
//     Drive/Inputs/In/nState1 @bit 1 <-> STM Status/Status/Ready
//     Drive/Inputs/In/nState1 <-> STM Status/Status/Ready to enable
//     Drive/Inputs/In/nState1 @bit 6 <-> STM Status/Status/Torque reduced
//     Drive/Inputs/In/nState1 @bit 2 <-> STM Status/Status/Warning
//     Drive/Inputs/In/nState2 @bit 3 <-> STM Status/Status/Digital input 1
//     Drive/Inputs/In/nState2 @bit 4 <-> STM Status/Status/Digital input 2
//     Drive/Inputs/In/nState2 @bit 5 <-> STM Status/Status/Sync error
//     Drive/Inputs/In/nState2 @bit 7 <-> STM Status/Status/TxPDO Toggle
//     Drive/Inputs/In/nState4 @bit 1 <-> WcState/InputToggle
//     Drive/Inputs/In/nState4 <-> WcState/WcState
//     Drive/Outputs/Out/nCtrl1 <-> STM Control/Control/Enable
//     Drive/Outputs/Out/nCtrl1 @bit 2 <-> STM Control/Control/Reduce torque
//     Drive/Outputs/Out/nCtrl1 @bit 1 <-> STM Control/Control/Reset
//     Drive/Outputs/Out/nCtrl2 @bit 3 <-> STM Control/Control/Digital output 1
//     Drive/Outputs/Out/nDataOut2[0] <-> STM Velocity/Velocity
//   (this object) <-> Device 2 (EtherCAT)/B950-233-WALL-S-R01-DRL-03_SDS/EK1122_04_17/B950-233-K2S13-DRL-01/EL5101_05_03
//     Enc/Inputs/In/nDataIn1[0] <-> ENC Status compact/Counter value
//     Enc/Inputs/In/nDataIn2[0] <-> ENC Status compact/Latch value
//     Enc/Inputs/In/nState1 @bit 4 <-> ENC Status compact/Status/Counter overflow
//     Enc/Inputs/In/nState1 @bit 3 <-> ENC Status compact/Status/Counter underflow
//     Enc/Inputs/In/nState1 @bit 7 <-> ENC Status compact/Status/Extrapolation stall
//     Enc/Inputs/In/nState1 <-> ENC Status compact/Status/Latch C valid
//     Enc/Inputs/In/nState1 @bit 1 <-> ENC Status compact/Status/Latch extern valid
//     Enc/Inputs/In/nState1 @bit 6 <-> ENC Status compact/Status/Open circuit
//     Enc/Inputs/In/nState1 @bit 2 <-> ENC Status compact/Status/Set counter done
//     Enc/Inputs/In/nState1 @bit 5 <-> ENC Status compact/Status/Status of input status
//     Enc/Inputs/In/nState2 @bit 4 <-> ENC Status compact/Status/Status of extern latch
//     Enc/Inputs/In/nState2 <-> ENC Status compact/Status/Status of input A
//     Enc/Inputs/In/nState2 @bit 1 <-> ENC Status compact/Status/Status of input B
//     Enc/Inputs/In/nState2 @bit 2 <-> ENC Status compact/Status/Status of input C
//     Enc/Inputs/In/nState2 @bit 3 <-> ENC Status compact/Status/Status of input gate
//     Enc/Inputs/In/nState2 @bit 5 <-> ENC Status compact/Status/Sync error
//     Enc/Inputs/In/nState2 @bit 6 <-> ENC Status compact/Status/TxPDO State
//     Enc/Inputs/In/nState2 @bit 7 <-> ENC Status compact/Status/TxPDO Toggle
//     Enc/Inputs/In/nState4 @bit 1 <-> WcState/InputToggle
//     Enc/Inputs/In/nState4 <-> WcState/WcState
//     Enc/Outputs/Out/nCtrl1 <-> ENC Control compact/Control/Enable latch C
//     Enc/Outputs/Out/nCtrl1 @bit 3 <-> ENC Control compact/Control/Enable latch extern on negative edge
//     Enc/Outputs/Out/nCtrl1 @bit 1 <-> ENC Control compact/Control/Enable latch extern on positive edge
//     Enc/Outputs/Out/nCtrl1 @bit 2 <-> ENC Control compact/Control/Set counter
//     Enc/Outputs/Out/nDataOut1[0] <-> ENC Control compact/Set counter value
//   (this object) <-> Device 2 (EtherCAT)/B950-233-WALL-S-R01-DRL-03_SDS/EL7047_04_12
//     Drive/Inputs/In/nState1 @bit 3 <-> STM Status/Status/Error
//     Drive/Inputs/In/nState1 @bit 7 <-> STM Status/Status/Motor stall
//     Drive/Inputs/In/nState1 @bit 5 <-> STM Status/Status/Moving negative
//     Drive/Inputs/In/nState1 @bit 4 <-> STM Status/Status/Moving positive
//     Drive/Inputs/In/nState1 @bit 1 <-> STM Status/Status/Ready
//     Drive/Inputs/In/nState1 <-> STM Status/Status/Ready to enable
//     Drive/Inputs/In/nState1 @bit 6 <-> STM Status/Status/Torque reduced
//     Drive/Inputs/In/nState1 @bit 2 <-> STM Status/Status/Warning
//     Drive/Inputs/In/nState2 @bit 3 <-> STM Status/Status/Digital input 1
//     Drive/Inputs/In/nState2 @bit 4 <-> STM Status/Status/Digital input 2
//     Drive/Inputs/In/nState2 @bit 5 <-> STM Status/Status/Sync error
//     Drive/Inputs/In/nState2 @bit 7 <-> STM Status/Status/TxPDO Toggle
//     Drive/Inputs/In/nState4 @bit 1 <-> WcState/InputToggle
//     Drive/Inputs/In/nState4 <-> WcState/WcState
//     Drive/Outputs/Out/nCtrl1 <-> STM Control/Control/Enable
//     Drive/Outputs/Out/nCtrl1 @bit 2 <-> STM Control/Control/Reduce torque
//     Drive/Outputs/Out/nCtrl1 @bit 1 <-> STM Control/Control/Reset
//     Drive/Outputs/Out/nCtrl2 @bit 3 <-> STM Control/Control/Digital output 1
//     Drive/Outputs/Out/nDataOut2[0] <-> STM Velocity/Velocity
//   (this object) <-> Device 2 (EtherCAT)/B950-233-WALL-S-R01-DRL-01/EL5042_02_13
//     Enc/Inputs/In/nComState @bit 1 <-> WcState/InputToggle
//     Enc/Inputs/In/nComState <-> WcState/WcState
//     Enc/Inputs/In/nDataIn1 <-> FB Inputs Channel 1/Position
//     Enc/Inputs/In/nDataIn1 <-> FB Inputs Channel 2/Position
//     Enc/Inputs/In/nState1 @bit 12 <-> FB Inputs Channel 1/Status/Diag
//     Enc/Inputs/In/nState1 @bit 12 <-> FB Inputs Channel 2/Status/Diag
//     Enc/Inputs/In/nState1 @bit 1 <-> FB Inputs Channel 1/Status/Error
//     Enc/Inputs/In/nState1 @bit 1 <-> FB Inputs Channel 2/Status/Error
//     Enc/Inputs/In/nState1 @bit 14 <-> FB Inputs Channel 1/Status/Input cycle counter
//     Enc/Inputs/In/nState1 @bit 14 <-> FB Inputs Channel 2/Status/Input cycle counter
//     Enc/Inputs/In/nState1 @bit 2 <-> FB Inputs Channel 1/Status/Ready
//     Enc/Inputs/In/nState1 @bit 2 <-> FB Inputs Channel 2/Status/Ready
//     Enc/Inputs/In/nState1 @bit 13 <-> FB Inputs Channel 1/Status/TxPDO State
//     Enc/Inputs/In/nState1 @bit 13 <-> FB Inputs Channel 2/Status/TxPDO State
//     Enc/Inputs/In/nState1 <-> FB Inputs Channel 1/Status/Warning
//     Enc/Inputs/In/nState1 <-> FB Inputs Channel 2/Status/Warning
//   (this object) <-> Device 2 (EtherCAT)/B950-233-WALL-S-R01-DRL-01/EL7047_02_12
//     Drive/Inputs/In/nState1 @bit 3 <-> STM Status/Status/Error
//     Drive/Inputs/In/nState1 @bit 7 <-> STM Status/Status/Motor stall
//     Drive/Inputs/In/nState1 @bit 5 <-> STM Status/Status/Moving negative
//     Drive/Inputs/In/nState1 @bit 4 <-> STM Status/Status/Moving positive
//     Drive/Inputs/In/nState1 @bit 1 <-> STM Status/Status/Ready
//     Drive/Inputs/In/nState1 <-> STM Status/Status/Ready to enable
//     Drive/Inputs/In/nState1 @bit 6 <-> STM Status/Status/Torque reduced
//     Drive/Inputs/In/nState1 @bit 2 <-> STM Status/Status/Warning
//     Drive/Inputs/In/nState2 @bit 3 <-> STM Status/Status/Digital input 1
//     Drive/Inputs/In/nState2 @bit 4 <-> STM Status/Status/Digital input 2
//     Drive/Inputs/In/nState2 @bit 5 <-> STM Status/Status/Sync error
//     Drive/Inputs/In/nState2 @bit 7 <-> STM Status/Status/TxPDO Toggle
//     Drive/Inputs/In/nState4 @bit 1 <-> WcState/InputToggle
//     Drive/Inputs/In/nState4 <-> WcState/WcState
//     Drive/Outputs/Out/nCtrl1 <-> STM Control/Control/Enable
//     Drive/Outputs/Out/nCtrl1 @bit 2 <-> STM Control/Control/Reduce torque
//     Drive/Outputs/Out/nCtrl1 @bit 1 <-> STM Control/Control/Reset
//     Drive/Outputs/Out/nCtrl2 @bit 3 <-> STM Control/Control/Digital output 1
//     Drive/Outputs/Out/nDataOut2[0] <-> STM Velocity/Velocity
//   (this object) <-> Device 2 (EtherCAT)/B950-233-WALL-S-R01-DRL-01/EL7047_02_14
//     Drive/Inputs/In/nState1 @bit 3 <-> STM Status/Status/Error
//     Drive/Inputs/In/nState1 @bit 7 <-> STM Status/Status/Motor stall
//     Drive/Inputs/In/nState1 @bit 5 <-> STM Status/Status/Moving negative
//     Drive/Inputs/In/nState1 @bit 4 <-> STM Status/Status/Moving positive
//     Drive/Inputs/In/nState1 @bit 1 <-> STM Status/Status/Ready
//     Drive/Inputs/In/nState1 <-> STM Status/Status/Ready to enable
//     Drive/Inputs/In/nState1 @bit 6 <-> STM Status/Status/Torque reduced
//     Drive/Inputs/In/nState1 @bit 2 <-> STM Status/Status/Warning
//     Drive/Inputs/In/nState2 @bit 3 <-> STM Status/Status/Digital input 1
//     Drive/Inputs/In/nState2 @bit 4 <-> STM Status/Status/Digital input 2
//     Drive/Inputs/In/nState2 @bit 5 <-> STM Status/Status/Sync error
//     Drive/Inputs/In/nState2 @bit 7 <-> STM Status/Status/TxPDO Toggle
//     Drive/Inputs/In/nState4 @bit 1 <-> WcState/InputToggle
//     Drive/Inputs/In/nState4 <-> WcState/WcState
//     Drive/Outputs/Out/nCtrl1 <-> STM Control/Control/Enable
//     Drive/Outputs/Out/nCtrl1 @bit 2 <-> STM Control/Control/Reduce torque
//     Drive/Outputs/Out/nCtrl1 @bit 1 <-> STM Control/Control/Reset
//     Drive/Outputs/Out/nCtrl2 @bit 3 <-> STM Control/Control/Digital output 1
//     Drive/Outputs/Out/nDataOut2[0] <-> STM Velocity/Velocity
//   (this object) <-> Device 2 (EtherCAT)/B950-233-WALL-S-R01-DRL-01/EL5042_02_16
//     Enc/Inputs/In/nComState @bit 1 <-> WcState/InputToggle
//     Enc/Inputs/In/nComState <-> WcState/WcState
//     Enc/Inputs/In/nDataIn1 <-> FB Inputs Channel 1/Position
//     Enc/Inputs/In/nState1 @bit 12 <-> FB Inputs Channel 1/Status/Diag
//     Enc/Inputs/In/nState1 @bit 12 <-> FB Inputs Channel 2/Status/Diag
//     Enc/Inputs/In/nState1 @bit 1 <-> FB Inputs Channel 1/Status/Error
//     Enc/Inputs/In/nState1 @bit 1 <-> FB Inputs Channel 2/Status/Error
//     Enc/Inputs/In/nState1 @bit 14 <-> FB Inputs Channel 1/Status/Input cycle counter
//     Enc/Inputs/In/nState1 @bit 14 <-> FB Inputs Channel 2/Status/Input cycle counter
//     Enc/Inputs/In/nState1 @bit 2 <-> FB Inputs Channel 1/Status/Ready
//     Enc/Inputs/In/nState1 @bit 2 <-> FB Inputs Channel 2/Status/Ready
//     Enc/Inputs/In/nState1 @bit 13 <-> FB Inputs Channel 1/Status/TxPDO State
//     Enc/Inputs/In/nState1 @bit 13 <-> FB Inputs Channel 2/Status/TxPDO State
//     Enc/Inputs/In/nState1 <-> FB Inputs Channel 1/Status/Warning
//     Enc/Inputs/In/nState1 <-> FB Inputs Channel 2/Status/Warning
//   (this object) <-> Device 2 (EtherCAT)/B950-233-WALL-S-R01-DRL-01/EL7047_02_15
//     Drive/Inputs/In/nState1 @bit 3 <-> STM Status/Status/Error
//     Drive/Inputs/In/nState1 @bit 7 <-> STM Status/Status/Motor stall
//     Drive/Inputs/In/nState1 @bit 5 <-> STM Status/Status/Moving negative
//     Drive/Inputs/In/nState1 @bit 4 <-> STM Status/Status/Moving positive
//     Drive/Inputs/In/nState1 @bit 1 <-> STM Status/Status/Ready
//     Drive/Inputs/In/nState1 <-> STM Status/Status/Ready to enable
//     Drive/Inputs/In/nState1 @bit 6 <-> STM Status/Status/Torque reduced
//     Drive/Inputs/In/nState1 @bit 2 <-> STM Status/Status/Warning
//     Drive/Inputs/In/nState2 @bit 3 <-> STM Status/Status/Digital input 1
//     Drive/Inputs/In/nState2 @bit 4 <-> STM Status/Status/Digital input 2
//     Drive/Inputs/In/nState2 @bit 5 <-> STM Status/Status/Sync error
//     Drive/Inputs/In/nState2 @bit 7 <-> STM Status/Status/TxPDO Toggle
//     Drive/Inputs/In/nState4 @bit 1 <-> WcState/InputToggle
//     Drive/Inputs/In/nState4 <-> WcState/WcState
//     Drive/Outputs/Out/nCtrl1 <-> STM Control/Control/Enable
//     Drive/Outputs/Out/nCtrl1 @bit 2 <-> STM Control/Control/Reduce torque
//     Drive/Outputs/Out/nCtrl1 @bit 1 <-> STM Control/Control/Reset
//     Drive/Outputs/Out/nCtrl2 @bit 3 <-> STM Control/Control/Digital output 1
//     Drive/Outputs/Out/nDataOut2[0] <-> STM Velocity/Velocity
//   (this object) <-> Device 2 (EtherCAT)/B950-233-WALL-S-R01-DRL-01/EL7047_02_11
//     Drive/Inputs/In/nState1 @bit 3 <-> STM Status/Status/Error
//     Drive/Inputs/In/nState1 @bit 7 <-> STM Status/Status/Motor stall
//     Drive/Inputs/In/nState1 @bit 5 <-> STM Status/Status/Moving negative
//     Drive/Inputs/In/nState1 @bit 4 <-> STM Status/Status/Moving positive
//     Drive/Inputs/In/nState1 @bit 1 <-> STM Status/Status/Ready
//     Drive/Inputs/In/nState1 <-> STM Status/Status/Ready to enable
//     Drive/Inputs/In/nState1 @bit 6 <-> STM Status/Status/Torque reduced
//     Drive/Inputs/In/nState1 @bit 2 <-> STM Status/Status/Warning
//     Drive/Inputs/In/nState2 @bit 3 <-> STM Status/Status/Digital input 1
//     Drive/Inputs/In/nState2 @bit 4 <-> STM Status/Status/Digital input 2
//     Drive/Inputs/In/nState2 @bit 5 <-> STM Status/Status/Sync error
//     Drive/Inputs/In/nState2 @bit 7 <-> STM Status/Status/TxPDO Toggle
//     Drive/Inputs/In/nState4 @bit 1 <-> WcState/InputToggle
//     Drive/Inputs/In/nState4 <-> WcState/WcState
//     Drive/Outputs/Out/nCtrl1 <-> STM Control/Control/Enable
//     Drive/Outputs/Out/nCtrl1 @bit 2 <-> STM Control/Control/Reduce torque
//     Drive/Outputs/Out/nCtrl1 @bit 1 <-> STM Control/Control/Reset
//     Drive/Outputs/Out/nCtrl2 @bit 3 <-> STM Control/Control/Digital output 1
//     Drive/Outputs/Out/nDataOut2[0] <-> STM Velocity/Velocity
//   (this object) <-> Device 2 (EtherCAT)/BOX-01 Coupler (EK1100)/BOX-22 DET_ROT (EL5042)
//     Enc/Inputs/In/nComState @bit 1 <-> WcState/InputToggle
//     Enc/Inputs/In/nComState <-> WcState/WcState
//     Enc/Inputs/In/nDataIn1 <-> FB Inputs Channel 1/Position
//     Enc/Inputs/In/nState1 @bit 12 <-> FB Inputs Channel 1/Status/Diag
//     Enc/Inputs/In/nState1 @bit 1 <-> FB Inputs Channel 1/Status/Error
//     Enc/Inputs/In/nState1 @bit 14 <-> FB Inputs Channel 1/Status/Input cycle counter
//     Enc/Inputs/In/nState1 @bit 2 <-> FB Inputs Channel 1/Status/Ready
//     Enc/Inputs/In/nState1 @bit 13 <-> FB Inputs Channel 1/Status/TxPDO State
//     Enc/Inputs/In/nState1 <-> FB Inputs Channel 1/Status/Warning
//   (this object) <-> Device 2 (EtherCAT)/BOX-01 Coupler (EK1100)/BOX-23 DET_ROT (EL7047)
//     Drive/Inputs/In/nState1 @bit 3 <-> STM Status/Status/Error
//     Drive/Inputs/In/nState1 @bit 7 <-> STM Status/Status/Motor stall
//     Drive/Inputs/In/nState1 @bit 5 <-> STM Status/Status/Moving negative
//     Drive/Inputs/In/nState1 @bit 4 <-> STM Status/Status/Moving positive
//     Drive/Inputs/In/nState1 @bit 1 <-> STM Status/Status/Ready
//     Drive/Inputs/In/nState1 <-> STM Status/Status/Ready to enable
//     Drive/Inputs/In/nState1 @bit 6 <-> STM Status/Status/Torque reduced
//     Drive/Inputs/In/nState1 @bit 2 <-> STM Status/Status/Warning
//     Drive/Inputs/In/nState2 @bit 3 <-> STM Status/Status/Digital input 1
//     Drive/Inputs/In/nState2 @bit 4 <-> STM Status/Status/Digital input 2
//     Drive/Inputs/In/nState2 @bit 5 <-> STM Status/Status/Sync error
//     Drive/Inputs/In/nState2 @bit 7 <-> STM Status/Status/TxPDO Toggle
//     Drive/Inputs/In/nState4 @bit 1 <-> WcState/InputToggle
//     Drive/Inputs/In/nState4 <-> WcState/WcState
//     Drive/Outputs/Out/nCtrl1 <-> STM Control/Control/Enable
//     Drive/Outputs/Out/nCtrl1 @bit 2 <-> STM Control/Control/Reduce torque
//     Drive/Outputs/Out/nCtrl1 @bit 1 <-> STM Control/Control/Reset
//     Drive/Outputs/Out/nCtrl2 @bit 3 <-> STM Control/Control/Digital output 1
//     Drive/Outputs/Out/nDataOut2[0] <-> STM Velocity/Velocity
//   (this object) <-> Device 2 (EtherCAT)
//     BOX-01 Coupler (EK1100)/BOX-02 SFIN(EL1904)/Module 1 (FSOES)/RxPDO/FSOE <-> Rack#1A-01 Coupler (EK1100)/Rack#1A-02 SFIN (EL1918)/ConnectionInputs/Message_4 TxPDO
//     BOX-01 Coupler (EK1100)/BOX-02 SFIN(EL1904)/Module 1 (FSOES)/TxPDO/FSOE <-> Rack#1A-01 Coupler (EK1100)/Rack#1A-02 SFIN (EL1918)/ConnectionOutputs/Message_4 RxPDO
//     Rack#1A-01 Coupler (EK1100)/Rack#1A-02 SFIN (EL1918)/ConnectionInputs/Message_3 TxPDO <-> Rack#1A-01 Coupler (EK1100)/Rack#1A-03 SFOUT(EL2912)/Module 1 (FSOE)/FSoE Outputs/FSOE
//     Rack#1A-01 Coupler (EK1100)/Rack#1A-02 SFIN (EL1918)/ConnectionInputs/Message_4 TxPDO <-> BOX-01 Coupler (EK1100)/BOX-02 SFIN(EL1904)/Module 1 (FSOES)/RxPDO/FSOE
//     Rack#1A-01 Coupler (EK1100)/Rack#1A-02 SFIN (EL1918)/ConnectionInputs/Message_6 TxPDO <-> Rack#2B-01 Coupler (EK1100)/Rack#2B-06 SFIN (EL1918)/Module 1 (FSOE)/FSoE Outputs/FSOE
//     Rack#1A-01 Coupler (EK1100)/Rack#1A-02 SFIN (EL1918)/ConnectionOutputs/Message_3 RxPDO <-> Rack#1A-01 Coupler (EK1100)/Rack#1A-03 SFOUT(EL2912)/Module 1 (FSOE)/FSoE Inputs/FSOE
//     Rack#1A-01 Coupler (EK1100)/Rack#1A-02 SFIN (EL1918)/ConnectionOutputs/Message_4 RxPDO <-> BOX-01 Coupler (EK1100)/BOX-02 SFIN(EL1904)/Module 1 (FSOES)/TxPDO/FSOE
//     Rack#1A-01 Coupler (EK1100)/Rack#1A-02 SFIN (EL1918)/ConnectionOutputs/Message_6 RxPDO <-> Rack#2B-01 Coupler (EK1100)/Rack#2B-06 SFIN (EL1918)/Module 1 (FSOE)/FSoE Inputs/FSOE
//     Rack#1A-01 Coupler (EK1100)/Rack#1A-03 SFOUT(EL2912)/Module 1 (FSOE)/FSoE Inputs/FSOE <-> Rack#1A-01 Coupler (EK1100)/Rack#1A-02 SFIN (EL1918)/ConnectionOutputs/Message_3 RxPDO
//     Rack#1A-01 Coupler (EK1100)/Rack#1A-03 SFOUT(EL2912)/Module 1 (FSOE)/FSoE Outputs/FSOE <-> Rack#1A-01 Coupler (EK1100)/Rack#1A-02 SFIN (EL1918)/ConnectionInputs/Message_3 TxPDO
//     Rack#2B-01 Coupler (EK1100)/Rack#2B-06 SFIN (EL1918)/Module 1 (FSOE)/FSoE Inputs/FSOE <-> Rack#1A-01 Coupler (EK1100)/Rack#1A-02 SFIN (EL1918)/ConnectionOutputs/Message_6 RxPDO
//     Rack#2B-01 Coupler (EK1100)/Rack#2B-06 SFIN (EL1918)/Module 1 (FSOE)/FSoE Outputs/FSOE <-> Rack#1A-01 Coupler (EK1100)/Rack#1A-02 SFIN (EL1918)/ConnectionInputs/Message_6 TxPDO
//   qrix_motion Instance <-> Device 2 (EtherCAT)/B950-233-R03-DRL-01 (EK1200)/Term 141 (EL6692)
//     PlcTask Inputs/GVL_Interface.QRIX_VAC_VGC_03_CLOSED_LIMIT_SWITCH <-> IO Inputs/QRIX_VAC_VGC_03_CLOSED_LIMIT_SWITCH
//     PlcTask Inputs/GVL_Interface.QRIX_VAC_VGC_03_CL_CMD <-> IO Inputs/QRIX_VAC_VGC_03_CL_CMD
//     PlcTask Inputs/GVL_Interface.QRIX_VAC_VGC_03_OPEN_LIMIT_SWITCH <-> IO Inputs/QRIX_VAC_VGC_03_OPEN_LIMIT_SWITCH
//     PlcTask Inputs/GVL_Interface.QRIX_VAC_VGC_03_OP_CMD <-> IO Inputs/QRIX_VAC_VGC_03_OP_CMD
//     PlcTask Outputs/GVL_Interface.QRIX_MOT_SDS_MMS_H_BACKWARD_EN <-> IO Outputs/QRIX_MOT_SDS_MMS_H_BACKWARD_EN
//     PlcTask Outputs/GVL_Interface.QRIX_MOT_SDS_MMS_H_FORWARD_EN <-> IO Outputs/QRIX_MOT_SDS_MMS_H_FORWARD_EN
//     PlcTask Outputs/GVL_Interface.QRIX_MOT_SDS_MMS_H_RAW_ENC_CNTS <-> IO Outputs/QRIX_MOT_SDS_MMS_H_RAW_ENC_CNTS
//   qrix_motion Instance <-> Device 2 (EtherCAT)/B950-233-WALL-S-R01-DRL-01/EL1004_02_03
//     PlcTask Inputs/PRG_SSL.bLimitBackwardEnable <-> Channel 2/Input
//     PlcTask Inputs/PRG_SSL.bLimitForwardEnable <-> Channel 3/Input
//   qrix_motion Instance <-> Device 2 (EtherCAT)/B950-233-WALL-S-R01-DRL-01/EL1088_02_06
//     PlcTask Inputs/Main.M36.bLimitBackwardEnable <-> Channel 5/Input
//     PlcTask Inputs/Main.M37.bLimitBackwardEnable <-> Channel 1/Input
//     PlcTask Inputs/Main.M38.bLimitBackwardEnable <-> Channel 3/Input
//     PlcTask Inputs/Main.M36.bLimitForwardEnable <-> Channel 6/Input
//     PlcTask Inputs/Main.M37.bLimitForwardEnable <-> Channel 2/Input
//     PlcTask Inputs/Main.M38.bLimitForwardEnable <-> Channel 4/Input
//   qrix_motion Instance <-> Device 2 (EtherCAT)/B950-233-WALL-S-R01-DRL-01/EL5042_02_02
//     PlcTask Inputs/Main.M1.nRawEncoderULINT <-> FB Inputs Channel 1/Position
//     PlcTask Inputs/PRG_SSL.nRenishawAbsEncSlaveCounts <-> FB Inputs Channel 1/Position
//   qrix_motion Instance <-> Device 2 (EtherCAT)/B950-233-WALL-S-R01-DRL-01/EL5042_02_05 - LAS_VIS
//     PlcTask Inputs/Main.M36.nRawEncoderULINT <-> FB Inputs Channel 1/Position
//   qrix_motion Instance <-> Device 2 (EtherCAT)/B950-233-WALL-S-R01-DRL-01/EL5042_02_08 - LAS_D_V-H
//     PlcTask Inputs/Main.M37.nRawEncoderULINT <-> FB Inputs Channel 2/Position
//     PlcTask Inputs/Main.M38.nRawEncoderULINT <-> FB Inputs Channel 1/Position
//   qrix_motion Instance <-> Device 2 (EtherCAT)/B950-233-WALL-S-R01-DRL-01/EL5042_02_13
//     PlcTask Inputs/Main.M46.nRawEncoderULINT <-> FB Inputs Channel 1/Position
//     PlcTask Inputs/Main.M47.nRawEncoderULINT <-> FB Inputs Channel 2/Position
//   qrix_motion Instance <-> Device 2 (EtherCAT)/B950-233-WALL-S-R01-DRL-01/EL5042_02_16
//     PlcTask Inputs/Main.M48.nRawEncoderULINT <-> FB Inputs Channel 1/Position
//     PlcTask Inputs/Main.M49.nRawEncoderULINT <-> FB Inputs Channel 2/Position
//     PlcTask Inputs/PRG_Cryo.stCryoRotEnc.Count <-> FB Inputs Channel 2/Position
//   qrix_motion Instance <-> Device 2 (EtherCAT)/B950-233-WALL-S-R01-DRL-01/EL7047_02_01 - SSL
//     PlcTask Inputs/Main.M1.bLimitBackwardEnable <-> STM Status/Status/Digital input 2
//     PlcTask Inputs/Main.M1.bLimitForwardEnable <-> STM Status/Status/Digital input 1
//   qrix_motion Instance <-> Device 2 (EtherCAT)/B950-233-WALL-S-R01-DRL-01/EL7047_02_11
//     PlcTask Inputs/PRG_Cryo.fbMeasureReferenceVelocityCryoROT.bCounterOverflow <-> ENC Status compact/Status/Counter overflow
//     PlcTask Inputs/PRG_Cryo.fbMeasureReferenceVelocityCryoROT.bCounterUnderflow <-> ENC Status compact/Status/Counter underflow
//     PlcTask Inputs/PRG_Cryo.fbMeasureReferenceVelocityCryoROT.nMicrostepCounter <-> ENC Status compact/Counter value
//     PlcTask Inputs/PRG_Cryo.stCryoRotDiffThetaCoordinateGantryAxisEnable.bFollowDriveReady <-> STM Status/Status/Ready
//   qrix_motion Instance <-> Device 2 (EtherCAT)/B950-233-WALL-S-R01-DRL-01/EL7047_02_12
//     PlcTask Inputs/Main.M46.bLimitBackwardEnable <-> STM Status/Status/Digital input 2
//     PlcTask Inputs/Main.M46.bLimitForwardEnable <-> STM Status/Status/Digital input 1
//     PlcTask Inputs/PRG_Cryo.fbMeasureReferenceVelocityCryoX.bCounterOverflow <-> ENC Status compact/Status/Counter overflow
//     PlcTask Inputs/PRG_Cryo.fbMeasureReferenceVelocityCryoX.bCounterUnderflow <-> ENC Status compact/Status/Counter underflow
//     PlcTask Inputs/PRG_Cryo.fbMeasureReferenceVelocityCryoX.nMicrostepCounter <-> ENC Status compact/Counter value
//     PlcTask Inputs/PRG_Cryo.stCryoXMultiLeader.bFollowerDriveReady <-> STM Status/Status/Ready
//   qrix_motion Instance <-> Device 2 (EtherCAT)/B950-233-WALL-S-R01-DRL-01/EL7047_02_14
//     PlcTask Inputs/Main.M47.bLimitBackwardEnable <-> STM Status/Status/Digital input 1
//     PlcTask Inputs/Main.M47.bLimitForwardEnable <-> STM Status/Status/Digital input 2
//     PlcTask Inputs/PRG_Cryo.fbMeasureReferenceVelocityCryoY.bCounterOverflow <-> ENC Status compact/Status/Counter overflow
//     PlcTask Inputs/PRG_Cryo.fbMeasureReferenceVelocityCryoY.bCounterUnderflow <-> ENC Status compact/Status/Counter underflow
//     PlcTask Inputs/PRG_Cryo.fbMeasureReferenceVelocityCryoY.nMicrostepCounter <-> ENC Status compact/Counter value
//     PlcTask Inputs/PRG_Cryo.stCryoYMultiLeader.bFollowerDriveReady <-> STM Status/Status/Ready
//   qrix_motion Instance <-> Device 2 (EtherCAT)/B950-233-WALL-S-R01-DRL-01/EL7047_02_15
//     PlcTask Inputs/Main.M48.bLimitBackwardEnable <-> STM Status/Status/Digital input 2
//     PlcTask Inputs/Main.M48.bLimitForwardEnable <-> STM Status/Status/Digital input 1
//     PlcTask Inputs/PRG_Cryo.fbMeasureReferenceVelocityCryoZ.bCounterOverflow <-> ENC Status compact/Status/Counter overflow
//     PlcTask Inputs/PRG_Cryo.fbMeasureReferenceVelocityCryoZ.bCounterUnderflow <-> ENC Status compact/Status/Counter underflow
//     PlcTask Inputs/PRG_Cryo.fbMeasureReferenceVelocityCryoZ.nMicrostepCounter <-> ENC Status compact/Counter value
//     PlcTask Inputs/PRG_Cryo.stCryoZMultiLeader.bFollowerDriveReady <-> STM Status/Status/Ready
//   qrix_motion Instance <-> Device 2 (EtherCAT)/B950-233-WALL-S-R01-DRL-02/EL1088_03_04
//     PlcTask Inputs/Main.M28.bLimitBackwardEnable <-> Channel 1/Input
//     PlcTask Inputs/Main.M29.bLimitBackwardEnable <-> Channel 3/Input
//     PlcTask Inputs/Main.M28.bLimitForwardEnable <-> Channel 2/Input
//     PlcTask Inputs/Main.M29.bLimitForwardEnable <-> Channel 4/Input
//   qrix_motion Instance <-> Device 2 (EtherCAT)/B950-233-WALL-S-R01-DRL-02/EL1088_03_08
//     PlcTask Inputs/Main.M30.bLimitBackwardEnable <-> Channel 1/Input
//     PlcTask Inputs/Main.M31.bLimitBackwardEnable <-> Channel 6/Input
//     PlcTask Inputs/Main.M32.bLimitBackwardEnable <-> Channel 4/Input
//     PlcTask Inputs/Main.M30.bLimitForwardEnable <-> Channel 2/Input
//     PlcTask Inputs/Main.M31.bLimitForwardEnable <-> Channel 5/Input
//     PlcTask Inputs/Main.M32.bLimitForwardEnable <-> Channel 3/Input
//   qrix_motion Instance <-> Device 2 (EtherCAT)/B950-233-WALL-S-R01-DRL-02/EL1088_03_10
//     PlcTask Inputs/Main.M28.bHome <-> Channel 1/Input
//     PlcTask Inputs/Main.M29.bHome <-> Channel 2/Input
//     PlcTask Inputs/Main.M30.bHome <-> Channel 3/Input
//     PlcTask Inputs/Main.M31.bHome <-> Channel 4/Input
//     PlcTask Inputs/Main.M32.bHome <-> Channel 4/Input
//     PlcTask Inputs/Main.M33.bHome <-> Channel 6/Input
//     PlcTask Inputs/Main.M34.bHome <-> Channel 7/Input
//     PlcTask Inputs/Main.M35.bHome <-> Channel 8/Input
//   qrix_motion Instance <-> Device 2 (EtherCAT)/B950-233-WALL-S-R01-DRL-02/EL1088_03_15
//     PlcTask Inputs/Main.M33.bLimitBackwardEnable <-> Channel 1/Input
//     PlcTask Inputs/Main.M34.bLimitBackwardEnable <-> Channel 4/Input
//     PlcTask Inputs/Main.M35.bLimitBackwardEnable <-> Channel 6/Input
//     PlcTask Inputs/Main.M33.bLimitForwardEnable <-> Channel 2/Input
//     PlcTask Inputs/Main.M34.bLimitForwardEnable <-> Channel 3/Input
//     PlcTask Inputs/Main.M35.bLimitForwardEnable <-> Channel 5/Input
//   qrix_motion Instance <-> Device 2 (EtherCAT)/B950-233-WALL-S-R01-DRL-02/EL5042_03_02-Diff-X-Y
//     PlcTask Inputs/Main.M28.nRawEncoderULINT <-> FB Inputs Channel 1/Position
//     PlcTask Inputs/Main.M29.nRawEncoderULINT <-> FB Inputs Channel 2/Position
//   qrix_motion Instance <-> Device 2 (EtherCAT)/B950-233-WALL-S-R01-DRL-02/EL5042_03_06-DIff-Z-2ThetaY
//     PlcTask Inputs/Main.M30.nRawEncoderULINT <-> FB Inputs Channel 1/Position
//     PlcTask Inputs/Main.M31.nRawEncoderULINT <-> FB Inputs Channel 2/Position
//   qrix_motion Instance <-> Device 2 (EtherCAT)/B950-233-WALL-S-R01-DRL-02/EL5042_03_13 - Diff - Phi - Chi
//     PlcTask Inputs/Main.M32.nRawEncoderULINT <-> FB Inputs Channel 1/Position
//     PlcTask Inputs/Main.M33.nRawEncoderULINT <-> FB Inputs Channel 2/Position
//   qrix_motion Instance <-> Device 2 (EtherCAT)/B950-233-WALL-S-R01-DRL-02/EL5042_03_17 - Diff - Theta - 2Theta
//     PlcTask Inputs/Main.M34.nRawEncoderULINT <-> FB Inputs Channel 1/Position
//     PlcTask Inputs/Main.M35.nRawEncoderULINT <-> FB Inputs Channel 2/Position
//     PlcTask Inputs/PRG_Cryo.stDiffThetaEnc.Count <-> FB Inputs Channel 1/Position
//   qrix_motion Instance <-> Device 2 (EtherCAT)/B950-233-WALL-S-R01-DRL-02/EL7047_03_16 - Diff - Theta
//     PlcTask Inputs/PRG_Cryo.stCryoRotDiffThetaCoordinateGantryAxisEnable.bLeaderDriveReady <-> STM Status/Status/Ready
//   qrix_motion Instance <-> Device 2 (EtherCAT)/B950-233-WALL-S-R01-DRL-03_SDS/EK1122_04_17/B950-233-K2S13-DRL-01/EL5101_05_01
//     PlcTask Inputs/Main.M42.nRawEncoderUINT <-> ENC Status compact/Counter value
//   qrix_motion Instance <-> Device 2 (EtherCAT)/B950-233-WALL-S-R01-DRL-03_SDS/EK1122_04_17/B950-233-K2S13-DRL-01/EL5101_05_02
//     PlcTask Inputs/Main.M43.nRawEncoderUINT <-> ENC Status compact/Counter value
//   qrix_motion Instance <-> Device 2 (EtherCAT)/B950-233-WALL-S-R01-DRL-03_SDS/EK1122_04_17/B950-233-K2S13-DRL-01/EL5101_05_03
//     PlcTask Inputs/Main.M44.nRawEncoderUINT <-> ENC Status compact/Counter value
//   qrix_motion Instance <-> Device 2 (EtherCAT)/B950-233-WALL-S-R01-DRL-03_SDS/EL1004_04_04
//     PlcTask Inputs/Main.M{39..42}.bHome <-> Channel {1..4}/Input  (4 links)
//   qrix_motion Instance <-> Device 2 (EtherCAT)/B950-233-WALL-S-R01-DRL-03_SDS/EL1004_04_09
//     PlcTask Inputs/Main.M43.bHome <-> Channel 1/Input
//     PlcTask Inputs/Main.M44.bHome <-> Channel 3/Input
//   qrix_motion Instance <-> Device 2 (EtherCAT)/B950-233-WALL-S-R01-DRL-03_SDS/EL5042_04_02
//     PlcTask Inputs/Main.M39.nRawEncoderULINT <-> FB Inputs Channel 1/Position
//     PlcTask Inputs/Main.M40.nRawEncoderULINT <-> FB Inputs Channel 2/Position
//   qrix_motion Instance <-> Device 2 (EtherCAT)/B950-233-WALL-S-R01-DRL-03_SDS/EL5042_04_06
//     PlcTask Inputs/Main.M41.nRawEncoderULINT <-> FB Inputs Channel 1/Position
//   qrix_motion Instance <-> Device 2 (EtherCAT)/B950-233-WALL-S-R01-DRL-03_SDS/EL7047_04_01
//     PlcTask Inputs/Main.M39.bLimitBackwardEnable <-> STM Status/Status/Digital input 2
//     PlcTask Inputs/Main.M39.bLimitForwardEnable <-> STM Status/Status/Digital input 1
//   qrix_motion Instance <-> Device 2 (EtherCAT)/B950-233-WALL-S-R01-DRL-03_SDS/EL7047_04_03
//     PlcTask Inputs/Main.M40.bLimitBackwardEnable <-> STM Status/Status/Digital input 1
//     PlcTask Inputs/Main.M40.bLimitForwardEnable <-> STM Status/Status/Digital input 2
//   qrix_motion Instance <-> Device 2 (EtherCAT)/B950-233-WALL-S-R01-DRL-03_SDS/EL7047_04_05
//     PlcTask Inputs/Main.M41.bLimitBackwardEnable <-> STM Status/Status/Digital input 2
//     PlcTask Inputs/Main.M41.bLimitForwardEnable <-> STM Status/Status/Digital input 1
//   qrix_motion Instance <-> Device 2 (EtherCAT)/B950-233-WALL-S-R01-DRL-03_SDS/EL7047_04_10
//     PlcTask Inputs/Main.M43.bLimitBackwardEnable <-> STM Status/Status/Digital input 1
//     PlcTask Inputs/Main.M43.bLimitForwardEnable <-> STM Status/Status/Digital input 2
//   qrix_motion Instance <-> Device 2 (EtherCAT)/B950-233-WALL-S-R01-DRL-03_SDS/EL7047_04_12
//     PlcTask Inputs/Main.M44.bLimitBackwardEnable <-> STM Status/Status/Digital input 2
//     PlcTask Inputs/Main.M44.bLimitForwardEnable <-> STM Status/Status/Digital input 1
//   qrix_motion Instance <-> Device 2 (EtherCAT)/BOX-01 Coupler (EK1100)/BOX-03 ENC_X1_X2 (EL5042)
//     PlcTask Inputs/Main.M18.nRawEncoderULINT <-> FB Inputs Channel 1/Position
//     PlcTask Inputs/Main.M19.nRawEncoderULINT <-> FB Inputs Channel 2/Position
//   qrix_motion Instance <-> Device 2 (EtherCAT)/BOX-01 Coupler (EK1100)/BOX-04 ENC_Y1_Y2 (EL5042)
//     PlcTask Inputs/Main.M20.nRawEncoderULINT <-> FB Inputs Channel 1/Position
//     PlcTask Inputs/Main.M21.nRawEncoderULINT <-> FB Inputs Channel 1/Position
//   qrix_motion Instance <-> Device 2 (EtherCAT)/BOX-01 Coupler (EK1100)/BOX-05 ENC_XDC_RyDC (EL5042)
//     PlcTask Inputs/Main.M22.nRawEncoderULINT <-> FB Inputs Channel 1/Position
//     PlcTask Inputs/Main.M23.nRawEncoderULINT <-> FB Inputs Channel 2/Position
//   qrix_motion Instance <-> Device 2 (EtherCAT)/BOX-01 Coupler (EK1100)/BOX-06 ENC_ZDC_YF1 (EL5042)
//     PlcTask Inputs/Main.M24.nRawEncoderULINT <-> FB Inputs Channel 1/Position
//     PlcTask Inputs/Main.M25.nRawEncoderULINT <-> FB Inputs Channel 2/Position
//     PlcTask Inputs/PRG_DET_ARM.stRenishawAbsEncMaster.Count <-> FB Inputs Channel 2/Position
//   qrix_motion Instance <-> Device 2 (EtherCAT)/BOX-01 Coupler (EK1100)/BOX-07 ENC_YF2_ZF (EL5042)
//     PlcTask Inputs/Main.M26.nRawEncoderULINT <-> FB Inputs Channel 1/Position
//     PlcTask Inputs/Main.M27.nRawEncoderULINT <-> FB Inputs Channel 2/Position
//     PlcTask Inputs/PRG_DET_ARM.stRenishawAbsEncSlave.Count <-> FB Inputs Channel 1/Position
//   qrix_motion Instance <-> Device 2 (EtherCAT)/BOX-01 Coupler (EK1100)/BOX-08 CP_SDC (EL9221-5000)
//     PlcTask Inputs/GVL_VAR.bCircuitBreakerB0108Tripped <-> OCP Inputs/Status/Tripped
//     PlcTask Outputs/GVL_VAR.bCircuitBreakerB0108Reset <-> OCP Outputs/Control/Reset
//   qrix_motion Instance <-> Device 2 (EtherCAT)/BOX-01 Coupler (EK1100)/BOX-09 DR_XSDC1 (EL7041-0052)
//     PlcTask Inputs/Main.M18.bLimitBackwardEnable <-> STM Status/Status/Digital input 2
//     PlcTask Inputs/Main.M18.bLimitForwardEnable <-> STM Status/Status/Digital input 1
//   qrix_motion Instance <-> Device 2 (EtherCAT)/BOX-01 Coupler (EK1100)/BOX-10 DR_XSDC2 (EL7041-0052)
//     PlcTask Inputs/Main.M19.bLimitBackwardEnable <-> STM Status/Status/Digital input 2
//     PlcTask Inputs/Main.M19.bLimitForwardEnable <-> STM Status/Status/Digital input 1
//   qrix_motion Instance <-> Device 2 (EtherCAT)/BOX-01 Coupler (EK1100)/BOX-11 DR_YSDC1 (EL7041-0052)
//     PlcTask Inputs/Main.M20.bLimitBackwardEnable <-> STM Status/Status/Digital input 2
//     PlcTask Inputs/Main.M20.bLimitForwardEnable <-> STM Status/Status/Digital input 1
//   qrix_motion Instance <-> Device 2 (EtherCAT)/BOX-01 Coupler (EK1100)/BOX-12 DR_YSDC2 (EL7041-0052)
//     PlcTask Inputs/Main.M21.bLimitBackwardEnable <-> STM Status/Status/Digital input 2
//     PlcTask Inputs/Main.M21.bLimitForwardEnable <-> STM Status/Status/Digital input 1
//   qrix_motion Instance <-> Device 2 (EtherCAT)/BOX-01 Coupler (EK1100)/BOX-13 CP_DC (EL9221-5000)
//     PlcTask Inputs/GVL_VAR.bCircuitBreakerB0113Tripped <-> OCP Inputs/Status/Tripped
//     PlcTask Outputs/GVL_VAR.bCircuitBreakerB0113Reset <-> OCP Outputs/Control/Reset
//   qrix_motion Instance <-> Device 2 (EtherCAT)/BOX-01 Coupler (EK1100)/BOX-14 DR_XDC (EL7041-0052)
//     PlcTask Inputs/Main.M22.bLimitBackwardEnable <-> STM Status/Status/Digital input 2
//     PlcTask Inputs/Main.M22.bLimitForwardEnable <-> STM Status/Status/Digital input 1
//   qrix_motion Instance <-> Device 2 (EtherCAT)/BOX-01 Coupler (EK1100)/BOX-15 DR_RyDC (EL7041-0052)
//     PlcTask Inputs/Main.M23.bLimitBackwardEnable <-> STM Status/Status/Digital input 2
//     PlcTask Inputs/Main.M23.bLimitForwardEnable <-> STM Status/Status/Digital input 1
//   qrix_motion Instance <-> Device 2 (EtherCAT)/BOX-01 Coupler (EK1100)/BOX-16 DR_ZDC (EL7041-0052)
//     PlcTask Inputs/Main.M24.bLimitBackwardEnable <-> STM Status/Status/Digital input 2
//     PlcTask Inputs/Main.M24.bLimitForwardEnable <-> STM Status/Status/Digital input 1
//   qrix_motion Instance <-> Device 2 (EtherCAT)/BOX-01 Coupler (EK1100)/BOX-18 CP_YF1_YF2 (EL9221-5000)
//     PlcTask Inputs/GVL_VAR.bCircuitBreakerB0118Tripped <-> OCP Inputs/Status/Tripped
//     PlcTask Outputs/GVL_VAR.bCircuitBreakerB0118Reset <-> OCP Outputs/Control/Reset
//   qrix_motion Instance <-> Device 2 (EtherCAT)/BOX-01 Coupler (EK1100)/BOX-19 MB_YF1_YF2 (EL2602)
//     PlcTask Outputs/Main.M25.bBrakeRelease <-> Channel 1/Output
//     PlcTask Outputs/Main.M26.bBrakeRelease <-> Channel 2/Output
//   qrix_motion Instance <-> Device 2 (EtherCAT)/BOX-01 Coupler (EK1100)/BOX-20 DR_YF1 (EL7047)
//     PlcTask Inputs/PRG_DET_ARM.fbMeasureReferenceVelocity.bCounterOverflow <-> ENC Status compact/Status/Counter overflow
//     PlcTask Inputs/PRG_DET_ARM.fbMeasureReferenceVelocity.bCounterUnderflow <-> ENC Status compact/Status/Counter underflow
//     PlcTask Inputs/PRG_DET_ARM.fbMeasureReferenceVelocity.nMicrostepCounter <-> ENC Status compact/Counter value
//   qrix_motion Instance <-> Device 2 (EtherCAT)/BOX-01 Coupler (EK1100)/BOX-22 DET_ROT (EL5042)
//     PlcTask Inputs/Main.M45.nRawEncoderULINT <-> FB Inputs Channel 1/Position
//   qrix_motion Instance <-> Device 2 (EtherCAT)/Rack#1A-01 Coupler (EK1100)/Rack#1A-02 SFIN (EL1918)
//     PlcTask Inputs/GVL_EPS.bESTOP <-> StandardInputs/Standard Out Var 18
//     PlcTask Inputs/Main.M25.bLimitBackwardEnable <-> StandardInputs/Standard Out Var 11
//     PlcTask Inputs/Main.M26.bLimitBackwardEnable <-> StandardInputs/Standard Out Var 13
//     PlcTask Inputs/Main.M27.bLimitBackwardEnable <-> StandardInputs/Standard Out Var 15
//     PlcTask Inputs/Main.M25.bLimitForwardEnable <-> StandardInputs/Standard Out Var 10
//     PlcTask Inputs/Main.M26.bLimitForwardEnable <-> StandardInputs/Standard Out Var 12
//     PlcTask Inputs/Main.M27.bLimitForwardEnable <-> StandardInputs/Standard Out Var 14
//     PlcTask Outputs/PRG_SpetrometerArm.bEnaIclk <-> StandardOutputs/Standard In Var 2
//     PlcTask Outputs/PRG_SpetrometerArm.bEnaIclkErrAck <-> StandardOutputs/Standard In Var 1
//     PlcTask Outputs/PRG_SpetrometerArm.bEnaIclkRestartESTOP <-> StandardOutputs/Standard In Var 9
//   qrix_motion Instance <-> Device 2 (EtherCAT)/Rack#1A-01 Coupler (EK1100)/Rack#1A-04 DR_2Th (EL7047)
//     PlcTask Inputs/Main.M2.bLimitBackwardEnable <-> STM Status/Status/Digital input 2
//     PlcTask Inputs/Main.M2.bLimitForwardEnable <-> STM Status/Status/Digital input 1
//     PlcTask Inputs/PRG_2Theta.b2ThetaDriveReady <-> STM Status/Status/Ready
//   qrix_motion Instance <-> Device 2 (EtherCAT)/Rack#1A-01 Coupler (EK1100)/Rack#1A-05 MB_2Th (EL2602)
//     PlcTask Outputs/Main.M2.bBrakeRelease <-> Channel 1/Output
//   qrix_motion Instance <-> Device 2 (EtherCAT)/Rack#1A-01 Coupler (EK1100)/Rack#1A-06 ENC_2Th (EL5042)
//     PlcTask Inputs/Main.M2.nRawEncoderULINT <-> FB Inputs Channel 1/Position
//     PlcTask Inputs/PRG_SSL.stRenishawAbsEncMaster.Count <-> FB Inputs Channel 1/Position
//   qrix_motion Instance <-> Device 2 (EtherCAT)/Rack#2A-01 Coupler (EK1100)/Rack#2A-02 CP_SLIT (EL9221-5000)
//     PlcTask Inputs/GVL_VAR.bCircuitBreakerR2A02Tripped <-> OCP Inputs/Status/Tripped
//     PlcTask Outputs/GVL_VAR.bCircuitBreakerR2A02Reset <-> OCP Outputs/Control/Reset
//   qrix_motion Instance <-> Device 2 (EtherCAT)/Rack#2A-01 Coupler (EK1100)/Rack#2A-03 DR_XS1 (EL7041-0052)
//     PlcTask Inputs/Main.M3.bLimitBackwardEnable <-> STM Status/Status/Digital input 2
//     PlcTask Inputs/Main.M3.bLimitForwardEnable <-> STM Status/Status/Digital input 1
//   qrix_motion Instance <-> Device 2 (EtherCAT)/Rack#2A-01 Coupler (EK1100)/Rack#2A-04 DR_XS2 (EL7041-0052)
//     PlcTask Inputs/Main.M4.bLimitBackwardEnable <-> STM Status/Status/Digital input 2
//     PlcTask Inputs/Main.M4.bLimitForwardEnable <-> STM Status/Status/Digital input 1
//   qrix_motion Instance <-> Device 2 (EtherCAT)/Rack#2A-01 Coupler (EK1100)/Rack#2A-05 DR_YS1 (EL7041-0052)
//     PlcTask Inputs/Main.M5.bLimitBackwardEnable <-> STM Status/Status/Digital input 2
//     PlcTask Inputs/Main.M5.bLimitForwardEnable <-> STM Status/Status/Digital input 1
//   qrix_motion Instance <-> Device 2 (EtherCAT)/Rack#2A-01 Coupler (EK1100)/Rack#2A-06 DR_YS2 (EL7041-0052)
//     PlcTask Inputs/Main.M6.bLimitBackwardEnable <-> STM Status/Status/Digital input 2
//     PlcTask Inputs/Main.M6.bLimitForwardEnable <-> STM Status/Status/Digital input 1
//   qrix_motion Instance <-> Device 2 (EtherCAT)/Rack#2A-01 Coupler (EK1100)/Rack#2A-07 CP_G (EL9221-5000)
//     PlcTask Inputs/GVL_VAR.bCircuitBreakerR2A07Tripped <-> OCP Inputs/Status/Tripped
//     PlcTask Outputs/GVL_VAR.bCircuitBreakerR2A07Reset <-> OCP Outputs/Control/Reset
//   qrix_motion Instance <-> Device 2 (EtherCAT)/Rack#2A-01 Coupler (EK1100)/Rack#2A-08 DR_RxG (EL7041-0052)
//     PlcTask Inputs/Main.M10.bLimitBackwardEnable <-> STM Status/Status/Digital input 2
//     PlcTask Inputs/Main.M10.bLimitForwardEnable <-> STM Status/Status/Digital input 1
//   qrix_motion Instance <-> Device 2 (EtherCAT)/Rack#2A-01 Coupler (EK1100)/Rack#2A-09 DR_XG (EL7041-0052)
//     PlcTask Inputs/Main.M11.bLimitBackwardEnable <-> STM Status/Status/Digital input 2
//     PlcTask Inputs/Main.M11.bLimitForwardEnable <-> STM Status/Status/Digital input 1
//   qrix_motion Instance <-> Device 2 (EtherCAT)/Rack#2A-01 Coupler (EK1100)/Rack#2A-10 DR_YG1 (EL7041-0052)
//     PlcTask Inputs/Main.M7.bLimitBackwardEnable <-> STM Status/Status/Digital input 2
//     PlcTask Inputs/Main.M7.bLimitForwardEnable <-> STM Status/Status/Digital input 1
//   qrix_motion Instance <-> Device 2 (EtherCAT)/Rack#2A-01 Coupler (EK1100)/Rack#2A-11 DR_YG2 (EL7041-0052)
//     PlcTask Inputs/Main.M8.bLimitBackwardEnable <-> STM Status/Status/Digital input 2
//     PlcTask Inputs/Main.M8.bLimitForwardEnable <-> STM Status/Status/Digital input 1
//   qrix_motion Instance <-> Device 2 (EtherCAT)/Rack#2A-01 Coupler (EK1100)/Rack#2A-12 DR_YG3 (EL7041-0052)
//     PlcTask Inputs/Main.M9.bLimitBackwardEnable <-> STM Status/Status/Digital input 2
//     PlcTask Inputs/Main.M9.bLimitForwardEnable <-> STM Status/Status/Digital input 1
//   qrix_motion Instance <-> Device 2 (EtherCAT)/Rack#2A-01 Coupler (EK1100)/Rack#2A-13 CP_PM (EL9221-5000)
//     PlcTask Inputs/GVL_VAR.bCircuitBreakerR2A13Tripped <-> OCP Inputs/Status/Tripped
//     PlcTask Outputs/GVL_VAR.bCircuitBreakerR2A13Reset <-> OCP Outputs/Control/Reset
//   qrix_motion Instance <-> Device 2 (EtherCAT)/Rack#2A-01 Coupler (EK1100)/Rack#2A-14 DR_XPM1 (EL7041-0052)
//     PlcTask Inputs/Main.M12.bLimitBackwardEnable <-> STM Status/Status/Digital input 2
//     PlcTask Inputs/Main.M12.bLimitForwardEnable <-> STM Status/Status/Digital input 1
//   qrix_motion Instance <-> Device 2 (EtherCAT)/Rack#2A-01 Coupler (EK1100)/Rack#2A-15 DR_XPM2 (EL7041-0052)
//     PlcTask Inputs/Main.M13.bLimitBackwardEnable <-> STM Status/Status/Digital input 2
//     PlcTask Inputs/Main.M13.bLimitForwardEnable <-> STM Status/Status/Digital input 1
//   qrix_motion Instance <-> Device 2 (EtherCAT)/Rack#2A-01 Coupler (EK1100)/Rack#2A-16 DR_RzPM (EL7041-0052)
//     PlcTask Inputs/Main.M14.bLimitBackwardEnable <-> STM Status/Status/Digital input 2
//     PlcTask Inputs/Main.M14.bLimitForwardEnable <-> STM Status/Status/Digital input 1
//   qrix_motion Instance <-> Device 2 (EtherCAT)/Rack#2B-01 Coupler (EK1100)/Rack#2B-03 AI_TiltSensor (EL3174-0002)
//     PlcTask Inputs/GVL_Sensor.stFrameP.iRawCnts <-> AI Standard Channel 4/Value
//     PlcTask Inputs/GVL_Sensor.stFrameR.iRawCnts <-> AI Standard Channel 3/Value
//     PlcTask Inputs/GVL_Sensor.stGraniteP.iRawCnts <-> AI Standard Channel 2/Value
//     PlcTask Inputs/GVL_Sensor.stGraniteR.iRawCnts <-> AI Standard Channel 1/Value
//   qrix_motion Instance <-> Device 2 (EtherCAT)/Rack#2B-01 Coupler (EK1100)/Rack#2B-04 PS_P (EL3064)
//     PlcTask Inputs/GVL_Sensor.stPS1.iRawCnts <-> AI Standard Channel 1/Value
//     PlcTask Inputs/GVL_Sensor.stPS2.iRawCnts <-> AI Standard Channel 2/Value
//     PlcTask Inputs/GVL_Sensor.stPS3.iRawCnts <-> AI Standard Channel 3/Value
//   qrix_motion Instance <-> Device 2 (EtherCAT)/Rack#2B-01 Coupler (EK1100)/Rack#2B-05 SV_AIR (EL2004)
//     PlcTask Outputs/GVL_EPS.bOpenSV1 <-> Channel 1/Output
//     PlcTask Outputs/GVL_EPS.bOpenSV2 <-> Channel 2/Output
//   qrix_motion Instance <-> Device 2 (EtherCAT)/Rack#2B-01 Coupler (EK1100)/Rack#2B-07 ENC_X1_X2 (EL5042)
//     PlcTask Inputs/Main.M3.nRawEncoderULINT <-> FB Inputs Channel 1/Position
//     PlcTask Inputs/Main.M4.nRawEncoderULINT <-> FB Inputs Channel 2/Position
//   qrix_motion Instance <-> Device 2 (EtherCAT)/Rack#2B-01 Coupler (EK1100)/Rack#2B-08 ENC_Y1_Y2 (EL5042)
//     PlcTask Inputs/Main.M5.nRawEncoderULINT <-> FB Inputs Channel 1/Position
//     PlcTask Inputs/Main.M6.nRawEncoderULINT <-> FB Inputs Channel 1/Position
//   qrix_motion Instance <-> Device 2 (EtherCAT)/Rack#2B-01 Coupler (EK1100)/Rack#2B-09 ENC_RxG_XG (EL5042)
//     PlcTask Inputs/Main.M10.nRawEncoderULINT <-> FB Inputs Channel 1 compact/Position
//     PlcTask Inputs/Main.M11.nRawEncoderULINT <-> FB Inputs Channel 2/Position
//   qrix_motion Instance <-> Device 2 (EtherCAT)/Rack#2B-01 Coupler (EK1100)/Rack#2B-10 ENC_YG1_YG2 (EL5042)
//     PlcTask Inputs/Main.M7.nRawEncoderULINT <-> FB Inputs Channel 1/Position
//     PlcTask Inputs/Main.M8.nRawEncoderULINT <-> FB Inputs Channel 2/Position
//   qrix_motion Instance <-> Device 2 (EtherCAT)/Rack#2B-01 Coupler (EK1100)/Rack#2B-11 ENC_YG3_X1PM (EL5042)
//     PlcTask Inputs/Main.M12.nRawEncoderULINT <-> FB Inputs Channel 2/Position
//     PlcTask Inputs/Main.M9.nRawEncoderULINT <-> FB Inputs Channel 1/Position
//   qrix_motion Instance <-> Device 2 (EtherCAT)/Rack#2B-01 Coupler (EK1100)/Rack#2B-12 ENC_X2PM_RzPM (EL5042)
//     PlcTask Inputs/Main.M13.nRawEncoderULINT <-> FB Inputs Channel 1/Position
//     PlcTask Inputs/Main.M14.nRawEncoderULINT <-> FB Inputs Channel 2/Position
//   qrix_motion Instance <-> Device 2 (EtherCAT)/Rack#2B-01 Coupler (EK1100)/Rack#2B-14 CP_YDF (EL9221-5000)
//     PlcTask Inputs/GVL_VAR.bCircuitBreakerR2B14Tripped <-> OCP Inputs/Status/Tripped
//     PlcTask Outputs/GVL_VAR.bCircuitBreakerR2B14Reset <-> OCP Outputs/Control/Reset
//   qrix_motion Instance <-> Device 2 (EtherCAT)/Rack#2B-01 Coupler (EK1100)/Rack#2B-15 DR_YDF1 (EL7041-0052)
//     PlcTask Inputs/Main.M15.bLimitBackwardEnable <-> STM Status/Status/Digital input 2
//     PlcTask Inputs/Main.M15.bLimitForwardEnable <-> STM Status/Status/Digital input 1
//   qrix_motion Instance <-> Device 2 (EtherCAT)/Rack#2B-01 Coupler (EK1100)/Rack#2B-16 DR_YDF2 (EL7041-0052)
//     PlcTask Inputs/Main.M16.bLimitBackwardEnable <-> STM Status/Status/Digital input 2
//     PlcTask Inputs/Main.M16.bLimitForwardEnable <-> STM Status/Status/Digital input 1
//   qrix_motion Instance <-> Device 2 (EtherCAT)/Rack#2B-01 Coupler (EK1100)/Rack#2B-17 CP_YDF_ZF (EL9221-5000)
//     PlcTask Inputs/GVL_VAR.bCircuitBreakerR2B17Tripped <-> OCP Inputs/Status/Tripped
//     PlcTask Outputs/GVL_VAR.bCircuitBreakerR2B17Reset <-> OCP Outputs/Control/Reset
//   qrix_motion Instance <-> Device 2 (EtherCAT)/Rack#2B-01 Coupler (EK1100)/Rack#2B-18 MB_ZF (EL2602)
//     PlcTask Outputs/Main.M27.bBrakeRelease <-> Channel 1/Output
//   qrix_motion Instance <-> Device 2 (EtherCAT)/Rack#2B-01 Coupler (EK1100)/Rack#2B-19 DR_YDF3 (EL7041-0052)
//     PlcTask Inputs/Main.M17.bLimitBackwardEnable <-> STM Status/Status/Digital input 2
//     PlcTask Inputs/Main.M17.bLimitForwardEnable <-> STM Status/Status/Digital input 1
//   qrix_motion Instance <-> Device 2 (EtherCAT)/Rack#2D LinearGaugeAmp (SC-HG1-ETC)
//     PlcTask Inputs/GVL_Sensor.stHDF.iRawCnts <-> Process Data(In)  TxPDO-Map/Response Data Unit4
//     PlcTask Inputs/GVL_Sensor.stYDF1.iRawCnts <-> Process Data(In)  TxPDO-Map/Response Data Unit1
//     PlcTask Inputs/GVL_Sensor.stYDF2.iRawCnts <-> Process Data(In)  TxPDO-Map/Response Data Unit2
//     PlcTask Inputs/GVL_Sensor.stYDF3.iRawCnts <-> Process Data(In)  TxPDO-Map/Response Data Unit3
//     PlcTask Inputs/Main.M15.nRawEncoderULINT <-> Process Data(In)  TxPDO-Map/Response Data Unit1
//     PlcTask Inputs/Main.M16.nRawEncoderULINT <-> Process Data(In)  TxPDO-Map/Response Data Unit2
//     PlcTask Inputs/Main.M17.nRawEncoderULINT <-> Process Data(In)  TxPDO-Map/Response Data Unit3
//     PlcTask Outputs/PRG_Sensor.bSensorHeadNormalValueMode <-> Process Data(Out) RxPDO-Map/Normal Value Mode
//     PlcTask Outputs/PRG_Sensor.bSensorHeadValueMode <-> Process Data(Out) RxPDO-Map/Head Value Mode
//   qrix_motion Instance <-> NC-Task 1 SAF/Axes/M1 - SSL Sliding seal
//     PlcTask Inputs/Main.M1.Axis.NcToPlc <-> Outputs/ToPlc
//     PlcTask Outputs/Main.M1.Axis.PlcToNc <-> Inputs/FromPlc
//     PlcTask Outputs/PRG_SSL.EL7047_02_01_SSL_Status_to_NC <-> Drive/Inputs/In/nState1
//   qrix_motion Instance <-> NC-Task 1 SAF/Axes/M10 - RxG
//     PlcTask Inputs/Main.M10.Axis.NcToPlc <-> Outputs/ToPlc
//     PlcTask Outputs/Main.M10.Axis.PlcToNc <-> Inputs/FromPlc
//   qrix_motion Instance <-> NC-Task 1 SAF/Axes/M11 - XG
//     PlcTask Inputs/Main.M11.Axis.NcToPlc <-> Outputs/ToPlc
//     PlcTask Outputs/Main.M11.Axis.PlcToNc <-> Inputs/FromPlc
//   qrix_motion Instance <-> NC-Task 1 SAF/Axes/M12 - XPM1
//     PlcTask Inputs/Main.M12.Axis.NcToPlc <-> Outputs/ToPlc
//     PlcTask Outputs/Main.M12.Axis.PlcToNc <-> Inputs/FromPlc
//   qrix_motion Instance <-> NC-Task 1 SAF/Axes/M13 - XPM2
//     PlcTask Inputs/Main.M13.Axis.NcToPlc <-> Outputs/ToPlc
//     PlcTask Outputs/Main.M13.Axis.PlcToNc <-> Inputs/FromPlc
//   qrix_motion Instance <-> NC-Task 1 SAF/Axes/M14 - RzPM
//     PlcTask Inputs/Main.M14.Axis.NcToPlc <-> Outputs/ToPlc
//     PlcTask Outputs/Main.M14.Axis.PlcToNc <-> Inputs/FromPlc
//   qrix_motion Instance <-> NC-Task 1 SAF/Axes/M15 - YDF1
//     PlcTask Inputs/Main.M15.Axis.NcToPlc <-> Outputs/ToPlc
//     PlcTask Outputs/GVL_Sensor.nYDF1 <-> Enc/Inputs/In/nDataIn1[0]
//     PlcTask Outputs/Main.M15.Axis.PlcToNc <-> Inputs/FromPlc
//     PlcTask Outputs/PRG_DET_FRAME.bLinearGaugeYDF1Ready <-> Enc/Inputs/In/nState1 @bit 2
//   qrix_motion Instance <-> NC-Task 1 SAF/Axes/M16 - YDF2
//     PlcTask Inputs/Main.M16.Axis.NcToPlc <-> Outputs/ToPlc
//     PlcTask Outputs/GVL_Sensor.nYDF2 <-> Enc/Inputs/In/nDataIn1[0]
//     PlcTask Outputs/Main.M16.Axis.PlcToNc <-> Inputs/FromPlc
//     PlcTask Outputs/PRG_DET_FRAME.bLinearGaugeYDF2Ready <-> Enc/Inputs/In/nState1 @bit 2
//   qrix_motion Instance <-> NC-Task 1 SAF/Axes/M17 - YDF3
//     PlcTask Inputs/Main.M17.Axis.NcToPlc <-> Outputs/ToPlc
//     PlcTask Outputs/GVL_Sensor.nYDF3 <-> Enc/Inputs/In/nDataIn1[0]
//     PlcTask Outputs/Main.M17.Axis.PlcToNc <-> Inputs/FromPlc
//     PlcTask Outputs/PRG_DET_FRAME.bLinearGaugeYDF3Ready <-> Enc/Inputs/In/nState1 @bit 2
//   qrix_motion Instance <-> NC-Task 1 SAF/Axes/M18 - XSDC1
//     PlcTask Inputs/Main.M18.Axis.NcToPlc <-> Outputs/ToPlc
//     PlcTask Outputs/Main.M18.Axis.PlcToNc <-> Inputs/FromPlc
//   qrix_motion Instance <-> NC-Task 1 SAF/Axes/M19 - XSDC2
//     PlcTask Inputs/Main.M19.Axis.NcToPlc <-> Outputs/ToPlc
//     PlcTask Outputs/Main.M19.Axis.PlcToNc <-> Inputs/FromPlc
//   qrix_motion Instance <-> NC-Task 1 SAF/Axes/M2 - 2Theta Stepper
//     PlcTask Inputs/Main.M2.Axis.NcToPlc <-> Outputs/ToPlc
//     PlcTask Outputs/Main.M2.Axis.PlcToNc <-> Inputs/FromPlc
//   qrix_motion Instance <-> NC-Task 1 SAF/Axes/M20 - YSDC1
//     PlcTask Inputs/Main.M20.Axis.NcToPlc <-> Outputs/ToPlc
//     PlcTask Outputs/Main.M20.Axis.PlcToNc <-> Inputs/FromPlc
//   qrix_motion Instance <-> NC-Task 1 SAF/Axes/M21 - YSDC2
//     PlcTask Inputs/Main.M21.Axis.NcToPlc <-> Outputs/ToPlc
//     PlcTask Outputs/Main.M21.Axis.PlcToNc <-> Inputs/FromPlc
//   qrix_motion Instance <-> NC-Task 1 SAF/Axes/M22 - XDC
//     PlcTask Inputs/Main.M22.Axis.NcToPlc <-> Outputs/ToPlc
//     PlcTask Outputs/Main.M22.Axis.PlcToNc <-> Inputs/FromPlc
//   qrix_motion Instance <-> NC-Task 1 SAF/Axes/M23 - RyDC
//     PlcTask Inputs/Main.M23.Axis.NcToPlc <-> Outputs/ToPlc
//     PlcTask Outputs/Main.M23.Axis.PlcToNc <-> Inputs/FromPlc
//   qrix_motion Instance <-> NC-Task 1 SAF/Axes/M24 - ZDC
//     PlcTask Inputs/Main.M24.Axis.NcToPlc <-> Outputs/ToPlc
//     PlcTask Outputs/Main.M24.Axis.PlcToNc <-> Inputs/FromPlc
//   qrix_motion Instance <-> NC-Task 1 SAF/Axes/M25 - YF1
//     PlcTask Inputs/Main.M25.Axis.NcToPlc <-> Outputs/ToPlc
//     PlcTask Outputs/Main.M25.Axis.PlcToNc <-> Inputs/FromPlc
//   qrix_motion Instance <-> NC-Task 1 SAF/Axes/M26 - YF2
//     PlcTask Inputs/Main.M26.Axis.NcToPlc <-> Outputs/ToPlc
//     PlcTask Outputs/Main.M26.Axis.PlcToNc <-> Inputs/FromPlc
//   qrix_motion Instance <-> NC-Task 1 SAF/Axes/M27 - ZF
//     PlcTask Inputs/Main.M27.Axis.NcToPlc <-> Outputs/ToPlc
//     PlcTask Outputs/Main.M27.Axis.PlcToNc <-> Inputs/FromPlc
//   qrix_motion Instance <-> NC-Task 1 SAF/Axes/M28 - Diff X
//     PlcTask Inputs/Main.M28.Axis.NcToPlc <-> Outputs/ToPlc
//     PlcTask Outputs/Main.M28.Axis.PlcToNc <-> Inputs/FromPlc
//   qrix_motion Instance <-> NC-Task 1 SAF/Axes/M29 - Diff Y
//     PlcTask Inputs/Main.M29.Axis.NcToPlc <-> Outputs/ToPlc
//     PlcTask Outputs/Main.M29.Axis.PlcToNc <-> Inputs/FromPlc
//   qrix_motion Instance <-> NC-Task 1 SAF/Axes/M3 - XS1
//     PlcTask Inputs/Main.M3.Axis.NcToPlc <-> Outputs/ToPlc
//     PlcTask Outputs/Main.M3.Axis.PlcToNc <-> Inputs/FromPlc
//   qrix_motion Instance <-> NC-Task 1 SAF/Axes/M30 - Diff Z
//     PlcTask Inputs/Main.M30.Axis.NcToPlc <-> Outputs/ToPlc
//     PlcTask Outputs/Main.M30.Axis.PlcToNc <-> Inputs/FromPlc
//   qrix_motion Instance <-> NC-Task 1 SAF/Axes/M31 - Diff 2Theta Y
//     PlcTask Inputs/Main.M31.Axis.NcToPlc <-> Outputs/ToPlc
//     PlcTask Outputs/Main.M31.Axis.PlcToNc <-> Inputs/FromPlc
//   qrix_motion Instance <-> NC-Task 1 SAF/Axes/M32 - Diff Phi
//     PlcTask Inputs/Main.M32.Axis.NcToPlc <-> Outputs/ToPlc
//     PlcTask Outputs/Main.M32.Axis.PlcToNc <-> Inputs/FromPlc
//   qrix_motion Instance <-> NC-Task 1 SAF/Axes/M33 - Diff Chi
//     PlcTask Inputs/Main.M33.Axis.NcToPlc <-> Outputs/ToPlc
//     PlcTask Outputs/Main.M33.Axis.PlcToNc <-> Inputs/FromPlc
//   qrix_motion Instance <-> NC-Task 1 SAF/Axes/M34 - Diff Theta
//     PlcTask Inputs/Main.M34.Axis.NcToPlc <-> Outputs/ToPlc
//     PlcTask Outputs/Main.M34.Axis.PlcToNc <-> Inputs/FromPlc
//     PlcTask Outputs/PRG_Cryo.nDiffThetaOutEncoderCounts <-> Enc/Inputs/In/nDataIn1
//   qrix_motion Instance <-> NC-Task 1 SAF/Axes/M35 - Diff 2Theta
//     PlcTask Inputs/Main.M35.Axis.NcToPlc <-> Outputs/ToPlc
//     PlcTask Outputs/Main.M35.Axis.PlcToNc <-> Inputs/FromPlc
//   qrix_motion Instance <-> NC-Task 1 SAF/Axes/M36 - LAS VIS
//     PlcTask Inputs/Main.M36.Axis.NcToPlc <-> Outputs/ToPlc
//     PlcTask Outputs/Main.M36.Axis.PlcToNc <-> Inputs/FromPlc
//   qrix_motion Instance <-> NC-Task 1 SAF/Axes/M37 - LAS D H
//     PlcTask Inputs/Main.M37.Axis.NcToPlc <-> Outputs/ToPlc
//     PlcTask Outputs/Main.M37.Axis.PlcToNc <-> Inputs/FromPlc
//   qrix_motion Instance <-> NC-Task 1 SAF/Axes/M38 - LAS D V
//     PlcTask Inputs/Main.M38.Axis.NcToPlc <-> Outputs/ToPlc
//     PlcTask Outputs/Main.M38.Axis.PlcToNc <-> Inputs/FromPlc
//   qrix_motion Instance <-> NC-Task 1 SAF/Axes/M39 - SDS X
//     PlcTask Inputs/Main.M39.Axis.NcToPlc <-> Outputs/ToPlc
//     PlcTask Outputs/Main.M39.Axis.PlcToNc <-> Inputs/FromPlc
//   qrix_motion Instance <-> NC-Task 1 SAF/Axes/M4 - XS2
//     PlcTask Inputs/Main.M4.Axis.NcToPlc <-> Outputs/ToPlc
//     PlcTask Outputs/Main.M4.Axis.PlcToNc <-> Inputs/FromPlc
//   qrix_motion Instance <-> NC-Task 1 SAF/Axes/M40 - SDS Y
//     PlcTask Inputs/Main.M40.Axis.NcToPlc <-> Outputs/ToPlc
//     PlcTask Outputs/Main.M40.Axis.PlcToNc <-> Inputs/FromPlc
//   qrix_motion Instance <-> NC-Task 1 SAF/Axes/M41 - SDS Z
//     PlcTask Inputs/Main.M41.Axis.NcToPlc <-> Outputs/ToPlc
//     PlcTask Outputs/Main.M41.Axis.PlcToNc <-> Inputs/FromPlc
//   qrix_motion Instance <-> NC-Task 1 SAF/Axes/M42 - SDS Rot Garage
//     PlcTask Inputs/Main.M42.Axis.NcToPlc <-> Outputs/ToPlc
//     PlcTask Outputs/Main.M42.Axis.PlcToNc <-> Inputs/FromPlc
//   qrix_motion Instance <-> NC-Task 1 SAF/Axes/M43 -SDS Linear Rotary
//     PlcTask Inputs/Main.M43.Axis.NcToPlc <-> Outputs/ToPlc
//     PlcTask Outputs/Main.M43.Axis.PlcToNc <-> Inputs/FromPlc
//   qrix_motion Instance <-> NC-Task 1 SAF/Axes/M44 - SDS Linear Horizontal
//     PlcTask Inputs/Main.M44.Axis.NcToPlc <-> Outputs/ToPlc
//     PlcTask Outputs/Main.M44.Axis.PlcToNc <-> Inputs/FromPlc
//   qrix_motion Instance <-> NC-Task 1 SAF/Axes/M45 - DET ROT
//     PlcTask Inputs/Main.M45.Axis.NcToPlc <-> Outputs/ToPlc
//     PlcTask Outputs/Main.M45.Axis.PlcToNc <-> Inputs/FromPlc
//   qrix_motion Instance <-> NC-Task 1 SAF/Axes/M46 - CRYO X
//     PlcTask Inputs/Main.M46.Axis.NcToPlc <-> Outputs/ToPlc
//     PlcTask Outputs/Main.M46.Axis.PlcToNc <-> Inputs/FromPlc
//   qrix_motion Instance <-> NC-Task 1 SAF/Axes/M47 - CRYO Y
//     PlcTask Inputs/Main.M47.Axis.NcToPlc <-> Outputs/ToPlc
//     PlcTask Outputs/Main.M47.Axis.PlcToNc <-> Inputs/FromPlc
//   qrix_motion Instance <-> NC-Task 1 SAF/Axes/M48 - CRYO Z
//     PlcTask Inputs/Main.M48.Axis.NcToPlc <-> Outputs/ToPlc
//     PlcTask Outputs/Main.M48.Axis.PlcToNc <-> Inputs/FromPlc
//   qrix_motion Instance <-> NC-Task 1 SAF/Axes/M49 - CRYO ROT
//     PlcTask Inputs/Main.M49.Axis.NcToPlc <-> Outputs/ToPlc
//     PlcTask Outputs/Main.M49.Axis.PlcToNc <-> Inputs/FromPlc
//     PlcTask Outputs/PRG_Cryo.nCryoRotOutEncoderCounts <-> Enc/Inputs/In/nDataIn1
//   qrix_motion Instance <-> NC-Task 1 SAF/Axes/M5 - YS1
//     PlcTask Inputs/Main.M5.Axis.NcToPlc <-> Outputs/ToPlc
//     PlcTask Outputs/Main.M5.Axis.PlcToNc <-> Inputs/FromPlc
//   qrix_motion Instance <-> NC-Task 1 SAF/Axes/M6 - YS2
//     PlcTask Inputs/Main.M6.Axis.NcToPlc <-> Outputs/ToPlc
//     PlcTask Outputs/Main.M6.Axis.PlcToNc <-> Inputs/FromPlc
//   qrix_motion Instance <-> NC-Task 1 SAF/Axes/M7 - YG1
//     PlcTask Inputs/Main.M7.Axis.NcToPlc <-> Outputs/ToPlc
//     PlcTask Outputs/Main.M7.Axis.PlcToNc <-> Inputs/FromPlc
//   qrix_motion Instance <-> NC-Task 1 SAF/Axes/M8 - YG2
//     PlcTask Inputs/Main.M8.Axis.NcToPlc <-> Outputs/ToPlc
//     PlcTask Outputs/Main.M8.Axis.PlcToNc <-> Inputs/FromPlc
//   qrix_motion Instance <-> NC-Task 1 SAF/Axes/M9 - YG3
//     PlcTask Inputs/Main.M9.Axis.NcToPlc <-> Outputs/ToPlc
//     PlcTask Outputs/Main.M9.Axis.PlcToNc <-> Inputs/FromPlc
//   qrix_motion Instance <-> qrix_motion/qrix_motion Instance
//     PlcTask Inputs/PRG_2Theta.nSSLDriveStatus <-> PlcTask Outputs/PRG_SSL.EL7047_02_01_SSL_Status_to_NC
//     PlcTask Outputs/PRG_SSL.EL7047_02_01_SSL_Status_to_NC <-> PlcTask Inputs/PRG_2Theta.nSSLDriveStatus

CONFIGURATION qrix_motion
    RESOURCE PLC ON TwinCAT3
        TASK PlcTask(INTERVAL := T#10ms, PRIORITY := 20);
        PROGRAM PRG_1_PlcTask WITH PlcTask : PRG_1_PlcTask;
    END_RESOURCE
END_CONFIGURATION

// ---- DUTs/DUT_Sensor.TcDUT

TYPE DUT_Sensor :
STRUCT
    fCntsInEGU:			REAL;
    {attribute 'pytmc' := '
        pv: EU
        io: i
    '}
    sEGU:				STRING;
    sName:				STRING;
    {attribute 'pytmc' := '
        pv: VALUE
        io: i
    '}
    fValue:				REAL;
    {attribute 'pytmc' := '
        pv: RAWCOUNTS
        io: i
    '}
    iRawCnts AT %I*:	INT;
    iOffset:			INT;
END_STRUCT
END_TYPE

// ---- DUTs/DUT_SensorHGS.TcDUT

TYPE DUT_SensorHGS:
STRUCT
    fCntsInEGU:			REAL;
    {attribute 'pytmc' := '
        pv: EU
        io: i
    '}
    sEGU:				STRING;
    sName:				STRING;
    {attribute 'pytmc' := '
        pv: VALUE
        io: i
    '}
    fValue:				REAL;
    {attribute 'pytmc' := '
        pv: RAWCOUNTS
        io: i
    '}
    iRawCnts AT %I*:	DINT;
    iOffset:			DINT;
END_STRUCT
END_TYPE

// ---- DUTs/ENUM_LAS_VIS_States.TcDUT

{attribute 'qualified_only'}
TYPE ENUM_LAS_VIS_States :
(
    UNKNOWN := 0,
    Position7to24mm := 1,
    Position62to77mm := 2
) UINT;
END_TYPE

// ---- DUTs/E_DiffState.TcDUT

{attribute 'qualified_only'}
TYPE E_DiffState :
(
    UNKNOWN := 0,
    TRANSFER_ARM_INTERFACE,
    NOMINAL_POSITION
) UINT;
END_TYPE

// ---- DUTs/E_GantryEnableState.TcDUT

{attribute 'qualified_only'}
{attribute 'strict'}
TYPE E_GantryEnableState :
(
    STANDBY,
    ERROR,
    WAIT_FOR_FULLY_ENABLED,
    WAIT_FOR_READY_STATE,
    DELAY_FOR_MOVE_START
);
END_TYPE

// ---- DUTs/E_MultiLeaderMotionCoupling.TcDUT

{attribute 'qualified_only'}
{attribute 'strict'}
TYPE E_MultiLeaderMotionCoupling :
(
    STATE_STANDBY,
    STATE_WAIT_FOR_FOLLOWER_NOT_BUSY,
    STATE_WAIT_FOR_FOLLOWER_ENABLED,
    STATE_WAIT_FOR_FOLLOWER_READY,
    STATE_ENABLE_EXTERNAL_SETPOINT_GENERATOR,
    STATE_FOLLOWING_ACTIVE,
    STATE_DISABLE_EXTERNAL_SETPOINT_GENERATOR,
    STATE_ERROR,
    STATE_MONITOR_TARGET_WINDOW,
    STATE_HALT_MOTION
) UDINT;
END_TYPE

// ---- DUTs/E_RealignCoupleState.TcDUT

{attribute 'qualified_only'}
{attribute 'strict'}
TYPE E_RealignCoupleState :
(
    STANDBY,
    DECOUPLE_AXES,
    COMMAND_AXES_INTO_REALIGNMENT,
    WAIT_FOR_MOVE_START,
    RECOUPLE_AXES,
    CLEANUP,
    ERROR
);
END_TYPE

// ---- DUTs/E_SampleSlotStates.TcDUT

{attribute 'qualified_only'}
{attribute 'strict'}
TYPE E_SampleSlotStates :
(
    EMPTY,
    FULL,
    DISABLED
);
END_TYPE

// ---- DUTs/E_SDSFaceState.TcDUT

{attribute 'qualified_only'}
{attribute 'strict'}
TYPE E_SDSFaceState :
(
    UNKNOWN := 0,
    FACE_TRANSFER_ARM := 1,
    FACE_SIDE_PORT := 2
) UINT;
END_TYPE

// ---- DUTs/E_SDSGarageYStates.TcDUT

{attribute 'qualified_only'}
TYPE E_SDSGarageYStates :
(
    UNKNOWN := 0,
    T1 := 1,
    T2 := 2,
    T3 := 3,
    T4 := 4,
    M1 := 5,
    M2 := 6,
    M3 := 7,
    M4 := 8,
    B1 := 9,
    B2 := 10,
    B3 := 11,
    B4 := 12,
    RETRACTED := 13
) UINT;
END_TYPE

// ---- DUTs/E_SDSGarageRStates.TcDUT

{attribute 'qualified_only'}
TYPE E_SDSGarageRStates :
(
    UNKNOWN := 0,
    T1 := 1,
    T2 := 2,
    T3 := 3,
    T4 := 4,
    M1 := 5,
    M2 := 6,
    M3 := 7,
    M4 := 8,
    B1 := 9,
    B2 := 10,
    B3 := 11,
    B4 := 12,
    PREDICTED_HOME := 13
) UINT;
END_TYPE

// ---- DUTs/E_SDSSubstate.TcDUT

{attribute 'qualified_only'}
TYPE E_SDSSubstate :
(
    Inactive,
    Select_Desired_Action,
    Check_Can_Home_Garage,
    Home_Garage,
    Check_Can_Home_Transfer_Arm,
    Home_Transfer_Arm,
    Check_Can_Load_Arm_From_Garage,
    Load_Arm_from_Garage,
    Check_Can_Unload_Arm_to_Garage,
    Unload_Arm_to_Garage,
    Check_Can_Load_Unload_Garage_from_Port,
    Load_Unload_Garage_from_Port,
    Check_Can_Load_Diffractometer_from_Arm,
    Load_Diffractometer_from_Arm,
    Check_Can_Unload_Diffractometer_to_Arm,
    Unload_Diffractometer_to_Arm,
    Check_Can_Manual_Control,
    Manual_Control
) UINT;
END_TYPE

// ---- DUTs/E_SDSTransferArmHStates.TcDUT

{attribute 'qualified_only'}
{attribute 'strict'}
TYPE E_SDSTransferArmHStates :
(
    UNKNOWN := 0,
    RETRACTED,
    GARAGE_SAMPLE_REMOVAL,
    CONFIRM_GARAGE_EXTRACTION,
    CONFIRM_DIFF_EXTRACTION,
    DIFF_SAMPLE_EXTRACTION,
    GARAGE_SAMPLE_INSERTION,
    CONFIRM_GARAGE_INSERTION,
    CONFIRM_DIFF_INSERTION,
    DIFF_SAMPLE_INSERTION
) UINT;
END_TYPE

// ---- DUTs/E_SDSHomingState.TcDUT

{attribute 'qualified_only'}
{attribute 'strict'}
TYPE E_SDSHomingState :
(
    INIT := 0,
    WAIT_NOT_BUSY,
    TRIGGER_HOMING,
    WAIT_FOR_HOMED,
    HOMED
) UINT;
END_TYPE

// ---- DUTs/E_SDSSeqState.TcDUT

{attribute 'qualified_only'}
TYPE E_SDSSeqState :
(
    Inactive,
    Home_Transfer_Arm,
    Check_Garage_Height,
    Manually_Rotate_Garage_for_Clearance_to_Raise,
    Retract_Garage_1,
    Home_Garage,
    Move_Diffractometer_to_Load_Unload_Position,
    Confirm_Vacuum_Valve_Open,
    Select_Garage_Slot_for_Removal,
    Select_Garage_Slot_for_Loading,
    Garage_Face_Transfer_Arm,
    Rotate_Garage_for_Clearance_to_Lower,
    Move_Garage_to_Slot_Height,
    Prerotate_Transfer_Arm_for_Extraction,
    Prerotate_Transfer_Arm_for_Insertion,
    Extend_Transfer_Arm_for_Extraction,
    Extend_Transfer_Arm_for_Insertion,
    Extend_Transfer_Arm_for_Diffractometer_Extraction,
    Extend_Transfer_Arm_for_Diffractometer_Insertion,
    Screw_in_Half_Turn,
    Fine_Adjustment,
    Unscrew_Sample_from_Garage,
    Unscrew_Sample_from_Diffractometer,
    Screw_Sample_into_Garage,
    Screw_Sample_into_Diffractometer,
    Confirm_Extraction,
    Confirm_Insertion,
    Confirm_Diffractometer_Insertion,
    Confirm_Diffractometer_Extraction,
    Update_Sample_Database,
    Retract_Transfer_Arm,
    Rotate_Garage_for_Clearance_to_Raise,
    Retract_Garage_2,
    Return_Garage_to_Home
) UINT;
END_TYPE

// ---- DUTs/E_SDSState.TcDUT

{attribute 'qualified_only'}
{attribute 'strict'}
TYPE E_SDSState :
(
    Standby,
    Error,
    Operating
) UINT;
END_TYPE

// ---- DUTs/E_SDSTransferArmRStates.TcDUT

{attribute 'qualified_only'}
{attribute 'strict'}
TYPE E_SDSTransferArmRStates :
(
    UNKNOWN := 0,
    FULLY_CCW,
    PREROTATE_SAMPLE_REMOVAL,
    PREROTATE_SAMPLE_INSERTION,
    UNSCREW_FROM_GARAGE,
    UNSCREW_FROM_DIFF,
    SCREW_INTO_GARAGE,
    SCREW_INTO_DIFF,
    SCREW_IN_HALF_TURN
) UINT;
END_TYPE

// ---- DUTs/ST_AutoRealignCouple.TcDUT

TYPE ST_AutoRealignCouple :
STRUCT
    {attribute 'pytmc' := '
        pv: eState
        io: i
        field: DESC Gives the current coupling realignment state.
    '}
    eState: E_RealignCoupleState;
    {attribute 'pytmc' := '
        pv: bExecute
        io: io
        field: DESC Hold TRUE to run an automatic realignment sequence. FALSE to cancel.
    '}
    bExecute: BOOL;
    {attribute 'pytmc' := '
        pv: bExecuteCouple
        io: io
        field: DESC Write TRUE to couple axes.
    '}
    bExecuteCouple: BOOL;
    {attribute 'pytmc' := '
        pv: bExecuteDecouple
        io: io
        field: DESC Write FALSE to decouple axes.
    '}
    bExecuteDecouple: BOOL;
    {attribute 'pytmc' := '
        pv: fRealignSpeed
        io: io
        field: DESC The speed at which the axis will be moved when realigning.
    '}
    fRealignSpeed: LREAL;
    {attribute 'pytmc' := '
        pv: bCoupled
        io: i
        field: DESC TRUE if the axes are coupled. FALSE if they are not coupled.
    '}
    bCoupled: BOOL;
END_STRUCT
END_TYPE

// ---- DUTs/ST_CoordinateGantryAxisEnable.TcDUT

